LIN {X 0,Y 516.678,Z 319.494,A -85,B 0,C 180,E1 19152.315,E2 19152.315} C_VEL
LIN {X 0,Y 512.908,Z 316.647,A -85,B 0,C 180,E1 19150.24,E2 19150.24} C_VEL
LIN {X 0,Y 508.959,Z 312.336,A -85,B 0,C 180,E1 19148.207,E2 19148.207} C_VEL
LIN {X 0,Y 504.801,Z 309.238,A -85,B 0,C 180,E1 19146.294,E2 19146.294} C_VEL
LIN {X 0,Y 500.678,Z 304.761,A -85,B 0,C 180,E1 19144.449,E2 19144.449} C_VEL
LIN {X 0,Y 496.281,Z 301.328,A -85,B 0,C 180,E1 19142.687,E2 19142.687} C_VEL
LIN {X 0,Y 492.471,Z 297.218,A -85,B 0,C 180,E1 19141.176,E2 19141.176} C_VEL
LIN {X 0,Y 487.825,Z 293.173,A -85,B 0,C 180,E1 19139.452,E2 19139.452} C_VEL
LIN {X 0,Y 484.702,Z 289.843,A -85,B 0,C 180,E1 19138.318,E2 19138.318} C_VEL
LIN {X 0,Y 480.021,Z 285.689,A -85,B 0,C 180,E1 19136.7,E2 19136.7} C_VEL
LIN {X 0,Y 477.029,Z 282.466,A -85,B 0,C 180,E1 19135.676,E2 19135.676} C_VEL
LIN {X 0,Y 472.507,Z 278.285,A -85,B 0,C 180,E1 19134.195,E2 19134.195} C_VEL
LIN {X 0,Y 469.925,Z 275.379,A -85,B 0,C 180,E1 19133.338,E2 19133.338} C_VEL
LIN {X 0,Y 465.029,Z 270.655,A -85,B 0,C 180,E1 19131.803,E2 19131.803} C_VEL
LIN {X 0,Y 462.666,Z 268.183,A -85,B 0,C 180,E1 19131.079,E2 19131.079} C_VEL
LIN {X 0,Y 458.047,Z 263.498,A -85,B 0,C 180,E1 19129.676,E2 19129.676} C_VEL
LIN {X 0,Y 455.814,Z 261.137,A -85,B 0,C 180,E1 19128.992,E2 19128.992} C_VEL
LIN {X 0,Y 451.033,Z 256.164,A -85,B 0,C 180,E1 19127.581,E2 19127.581} C_VEL
LIN {X 0,Y 445.033,Z 249.934,A -85,B 0,C 180,E1 19125.861,E2 19125.861} C_VEL
LIN {X 0,Y 443.054,Z 247.797,A -85,B 0,C 180,E1 19125.308,E2 19125.308} C_VEL
LIN {X 0,Y 438.624,Z 243.367,A -85,B 0,C 180,E1 19124.141,E2 19124.141} C_VEL
LIN {X 0,Y 436.476,Z 241.078,A -85,B 0,C 180,E1 19123.594,E2 19123.594} C_VEL
LIN {X 0,Y 432.178,Z 236.724,A -85,B 0,C 180,E1 19122.544,E2 19122.544} C_VEL
LIN {X 0,Y 430.194,Z 234.427,A -85,B 0,C 180,E1 19122.065,E2 19122.065} C_VEL
LIN {X 0,Y 429.077,Z 233.472,A -85,B 0,C 180,E1 19121.812,E2 19121.812} C_VEL
LIN {X 0,Y 423.316,Z 229.525,A -85,B 0,C 180,E1 19120.566,E2 19120.566} C_VEL
LIN {X 0,Y 413.271,Z 224.33,A -85,B 0,C 180,E1 19118.597,E2 19118.597} C_VEL
LIN {X 0,Y 410.338,Z 222.17,A -85,B 0,C 180,E1 19118.018,E2 19118.018} C_VEL
LIN {X 0,Y 407.486,Z 218.551,A -85,B 0,C 180,E1 19117.396,E2 19117.396} C_VEL
LIN {X 0,Y 406.442,Z 216.882,A -85,B 0,C 180,E1 19117.154,E2 19117.154} C_VEL
LIN {X 0,Y 403.788,Z 214.24,A -85,B 0,C 180,E1 19116.574,E2 19116.574} C_VEL
LIN {X 0,Y 402.666,Z 211.461,A -85,B 0,C 180,E1 19116.164,E2 19116.164} C_VEL
LIN {X 0,Y 402.566,Z 210.942,A -85,B 0,C 180,E1 19115.455,E2 19115.455} C_VEL
LIN {X 0,Y 402.577,Z 211.024,A -85,B 0,C 180,E1 19111.592,E2 19111.592} C_VEL
LIN {X 0,Y 402.567,Z 210.925,A -85,B 0,C 180,E1 19107.676,E2 19107.676} C_VEL
LIN {X 0,Y 402.577,Z 211.022,A -85,B 0,C 180,E1 19103.726,E2 19103.726} C_VEL
LIN {X 0,Y 402.577,Z 211.018,A -85,B 0,C 180,E1 19099.742,E2 19099.742} C_VEL
LIN {X 0,Y 402.573,Z 211.002,A -85,B 0,C 180,E1 19095.856,E2 19095.856} C_VEL
LIN {X 0,Y 402.573,Z 210.991,A -85,B 0,C 180,E1 19091.897,E2 19091.897} C_VEL
LIN {X 0,Y 402.574,Z 210.995,A -85,B 0,C 180,E1 19087.995,E2 19087.995} C_VEL
LIN {X 0,Y 402.574,Z 211.015,A -85,B 0,C 180,E1 19083.988,E2 19083.988} C_VEL
LIN {X 0,Y 402.574,Z 211.02,A -85,B 0,C 180,E1 19080,E2 19080} C_VEL
LIN {X 0,Y 402.574,Z 210.997,A -85,B 0,C 180,E1 19076.012,E2 19076.012} C_VEL
LIN {X 0,Y 402.572,Z 210.987,A -85,B 0,C 180,E1 19072.148,E2 19072.148} C_VEL
LIN {X 0,Y 402.575,Z 211,A -85,B 0,C 180,E1 19068.248,E2 19068.248} C_VEL
LIN {X 0,Y 402.578,Z 211.02,A -85,B 0,C 180,E1 19064.292,E2 19064.292} C_VEL
LIN {X 0,Y 402.579,Z 211.022,A -85,B 0,C 180,E1 19060.409,E2 19060.409} C_VEL
LIN {X 0,Y 402.584,Z 211.009,A -85,B 0,C 180,E1 19056.585,E2 19056.585} C_VEL
LIN {X 0,Y 402.582,Z 210.933,A -85,B 0,C 180,E1 19052.753,E2 19052.753} C_VEL
LIN {X 0,Y 402.591,Z 210.985,A -85,B 0,C 180,E1 19048.896,E2 19048.896} C_VEL
LIN {X 0,Y 402.601,Z 211.025,A -85,B 0,C 180,E1 19045.032,E2 19045.032} C_VEL
LIN {X 0,Y 402.714,Z 211.75,A -85,B 0,C 180,E1 19044.654,E2 19044.654} C_VEL
LIN {X 0,Y 404.399,Z 215.495,A -85,B 0,C 180,E1 19043.6,E2 19043.6} C_VEL
LIN {X 0,Y 414.866,Z 230.627,A -85,B 0,C 180,E1 19041.263,E2 19041.263} C_VEL
LIN {X 0,Y 422.772,Z 242.404,A -85,B 0,C 180,E1 19039.651,E2 19039.651} C_VEL
LIN {X 0,Y 432.944,Z 258.691,A -85,B 0,C 180,E1 19037.706,E2 19037.706} C_VEL
LIN {X 0,Y 444.241,Z 278.519,A -85,B 0,C 180,E1 19035.686,E2 19035.686} C_VEL
LIN {X 0,Y 455.277,Z 300.15,A -85,B 0,C 180,E1 19033.824,E2 19033.824} C_VEL
LIN {X 0,Y 456.625,Z 303.478,A -85,B 0,C 180,E1 19033.592,E2 19033.592} C_VEL
LIN {X 0,Y 447.384,Z 520.785,A -85,B 0,C 180,E1 19030.062,E2 19030.062} C_VEL
LIN {X 0,Y 445.937,Z 538.911,A -85,B 0,C 180,E1 19029.651,E2 19029.651} C_VEL
LIN {X 0,Y 443.556,Z 560.38,A -85,B 0,C 180,E1 19028.986,E2 19028.986} C_VEL
LIN {X 0,Y 440.354,Z 582.229,A -85,B 0,C 180,E1 19028.054,E2 19028.054} C_VEL
LIN {X 0,Y 437.341,Z 599.726,A -85,B 0,C 180,E1 19027.121,E2 19027.121} C_VEL
LIN {X 0,Y 434.267,Z 615.592,A -85,B 0,C 180,E1 19026.111,E2 19026.111} C_VEL
LIN {X 0,Y 431.179,Z 630.152,A -85,B 0,C 180,E1 19025.028,E2 19025.028} C_VEL
LIN {X 0,Y 427.866,Z 644.6,A -85,B 0,C 180,E1 19023.787,E2 19023.787} C_VEL
LIN {X 0,Y 424.501,Z 658.489,A -85,B 0,C 180,E1 19022.412,E2 19022.412} C_VEL
LIN {X 0,Y 421.02,Z 672.173,A -85,B 0,C 180,E1 19020.858,E2 19020.858} C_VEL
LIN {X 0,Y 417.315,Z 686.298,A -85,B 0,C 180,E1 19019.008,E2 19019.008} C_VEL
LIN {X 0,Y 412.921,Z 702.744,A -85,B 0,C 180,E1 19016.455,E2 19016.455} C_VEL
LIN {X 0,Y 409.682,Z 714.914,A -85,B 0,C 180,E1 19014.203,E2 19014.203} C_VEL
LIN {X 0,Y 407.133,Z 724.889,A -85,B 0,C 180,E1 19012.068,E2 19012.068} C_VEL
LIN {X 0,Y 404.954,Z 733.96,A -85,B 0,C 180,E1 19009.822,E2 19009.822} C_VEL
LIN {X 0,Y 403.169,Z 742.134,A -85,B 0,C 180,E1 19007.46,E2 19007.46} C_VEL
LIN {X 0,Y 401.726,Z 749.741,A -85,B 0,C 180,E1 19004.852,E2 19004.852} C_VEL
LIN {X 0,Y 400.599,Z 757.452,A -85,B 0,C 180,E1 19001.517,E2 19001.517} C_VEL
LIN {X 0,Y 400.13,Z 762.218,A -85,B 0,C 180,E1 18998.767,E2 18998.767} C_VEL
LIN {X 0,Y 399.973,Z 765.375,A -85,B 0,C 180,E1 18996.314,E2 18996.314} C_VEL
LIN {X 0,Y 399.939,Z 767.492,A -85,B 0,C 180,E1 18993.87,E2 18993.87} C_VEL
LIN {X 0,Y 399.948,Z 768.59,A -85,B 0,C 180,E1 18991.432,E2 18991.432} C_VEL
LIN {X 0,Y 399.955,Z 768.708,A -85,B 0,C 180,E1 18989.141,E2 18989.141} C_VEL
LIN {X 0,Y 399.936,Z 767.846,A -85,B 0,C 180,E1 18986.704,E2 18986.704} C_VEL
LIN {X 0,Y 399.951,Z 765.967,A -85,B 0,C 180,E1 18984.262,E2 18984.262} C_VEL
LIN {X 0,Y 400.076,Z 762.997,A -85,B 0,C 180,E1 18981.773,E2 18981.773} C_VEL
LIN {X 0,Y 400.407,Z 759.074,A -85,B 0,C 180,E1 18979.352,E2 18979.352} C_VEL
LIN {X 0,Y 401.047,Z 753.989,A -85,B 0,C 180,E1 18976.888,E2 18976.888} C_VEL
LIN {X 0,Y 402.002,Z 748.142,A -85,B 0,C 180,E1 18974.568,E2 18974.568} C_VEL
LIN {X 0,Y 403.361,Z 741.196,A -85,B 0,C 180,E1 18972.25,E2 18972.25} C_VEL
LIN {X 0,Y 405.16,Z 733.067,A -85,B 0,C 180,E1 18969.941,E2 18969.941} C_VEL
LIN {X 0,Y 407.609,Z 723.032,A -85,B 0,C 180,E1 18967.504,E2 18967.504} C_VEL
LIN {X 0,Y 411.234,Z 709.077,A -85,B 0,C 180,E1 18964.667,E2 18964.667} C_VEL
LIN {X 0,Y 414.498,Z 696.788,A -85,B 0,C 180,E1 18962.569,E2 18962.569} C_VEL
LIN {X 0,Y 417.854,Z 684.221,A -85,B 0,C 180,E1 18960.706,E2 18960.706} C_VEL
LIN {X 0,Y 421.097,Z 671.876,A -85,B 0,C 180,E1 18959.106,E2 18959.106} C_VEL
LIN {X 0,Y 424.501,Z 658.492,A -85,B 0,C 180,E1 18957.588,E2 18957.588} C_VEL
LIN {X 0,Y 427.867,Z 644.6,A -85,B 0,C 180,E1 18956.213,E2 18956.213} C_VEL
LIN {X 0,Y 431.179,Z 630.151,A -85,B 0,C 180,E1 18954.972,E2 18954.972} C_VEL
LIN {X 0,Y 434.454,Z 614.671,A -85,B 0,C 180,E1 18953.825,E2 18953.825} C_VEL
LIN {X 0,Y 437.539,Z 598.663,A -85,B 0,C 180,E1 18952.817,E2 18952.817} C_VEL
LIN {X 0,Y 440.807,Z 579.508,A -85,B 0,C 180,E1 18951.812,E2 18951.812} C_VEL
LIN {X 0,Y 443.971,Z 556.629,A -85,B 0,C 180,E1 18950.887,E2 18950.887} C_VEL
LIN {X 0,Y 446.015,Z 538.025,A -85,B 0,C 180,E1 18950.326,E2 18950.326} C_VEL
LIN {X 0,Y 447.414,Z 520.27,A -85,B 0,C 180,E1 18949.928,E2 18949.928} C_VEL
LIN {X 0,Y 456.615,Z 302.923,A -85,B 0,C 180,E1 18946.395,E2 18946.395} C_VEL
LIN {X 0,Y 445.675,Z 281.186,A -85,B 0,C 180,E1 18944.561,E2 18944.561} C_VEL
LIN {X 0,Y 434.191,Z 260.787,A -85,B 0,C 180,E1 18942.524,E2 18942.524} C_VEL
LIN {X 0,Y 424.621,Z 245.292,A -85,B 0,C 180,E1 18940.714,E2 18940.714} C_VEL
LIN {X 0,Y 416.039,Z 232.351,A -85,B 0,C 180,E1 18938.983,E2 18938.983} C_VEL
LIN {X 0,Y 408.694,Z 221.675,A -85,B 0,C 180,E1 18937.399,E2 18937.399} C_VEL
LIN {X 0,Y 404.615,Z 215.942,A -85,B 0,C 180,E1 18936.465,E2 18936.465} C_VEL
LIN {X 0,Y 403.803,Z 214.337,A -85,B 0,C 180,E1 18936.11,E2 18936.11} C_VEL
LIN {X 0,Y 402.6,Z 211.068,A -85,B 0,C 180,E1 18935.09,E2 18935.09} C_VEL
LIN {X 0,Y 402.583,Z 210.994,A -85,B 0,C 180,E1 18931.272,E2 18931.272} C_VEL
LIN {X 0,Y 402.571,Z 210.93,A -85,B 0,C 180,E1 18927.515,E2 18927.515} C_VEL
LIN {X 0,Y 402.578,Z 211.013,A -85,B 0,C 180,E1 18923.6,E2 18923.6} C_VEL
LIN {X 0,Y 402.577,Z 211.019,A -85,B 0,C 180,E1 18919.742,E2 18919.742} C_VEL
LIN {X 0,Y 402.576,Z 211.012,A -85,B 0,C 180,E1 18915.856,E2 18915.856} C_VEL
LIN {X 0,Y 402.575,Z 210.997,A -85,B 0,C 180,E1 18911.897,E2 18911.897} C_VEL
LIN {X 0,Y 402.574,Z 210.989,A -85,B 0,C 180,E1 18907.995,E2 18907.995} C_VEL
LIN {X 0,Y 402.577,Z 211.003,A -85,B 0,C 180,E1 18904.131,E2 18904.131} C_VEL
LIN {X 0,Y 402.579,Z 211.021,A -85,B 0,C 180,E1 18900.285,E2 18900.285} C_VEL
LIN {X 0,Y 402.583,Z 211.003,A -85,B 0,C 180,E1 18896.44,E2 18896.44} C_VEL
LIN {X 0,Y 402.587,Z 210.991,A -85,B 0,C 180,E1 18892.58,E2 18892.58} C_VEL
LIN {X 0,Y 402.599,Z 210.996,A -85,B 0,C 180,E1 18888.779,E2 18888.779} C_VEL
LIN {X 0,Y 402.606,Z 211.014,A -85,B 0,C 180,E1 18884.884,E2 18884.884} C_VEL
LIN {X 0,Y 402.614,Z 211.016,A -85,B 0,C 180,E1 18881.014,E2 18881.014} C_VEL
LIN {X 0,Y 402.614,Z 211.007,A -85,B 0,C 180,E1 18877.051,E2 18877.051} C_VEL
LIN {X 0,Y 402.603,Z 210.927,A -85,B 0,C 180,E1 18873.127,E2 18873.127} C_VEL
LIN {X 0,Y 402.619,Z 210.988,A -85,B 0,C 180,E1 18869.222,E2 18869.222} C_VEL
LIN {X 0,Y 402.607,Z 210.937,A -85,B 0,C 180,E1 18865.279,E2 18865.279} C_VEL
LIN {X 0,Y 402.629,Z 211.28,A -85,B 0,C 180,E1 18863.91,E2 18863.91} C_VEL
LIN {X 0,Y 403.059,Z 212.799,A -85,B 0,C 180,E1 18863.615,E2 18863.615} C_VEL
LIN {X 0,Y 405.049,Z 215.794,A -85,B 0,C 180,E1 18863.14,E2 18863.14} C_VEL
LIN {X 0,Y 407.043,Z 217.67,A -85,B 0,C 180,E1 18862.711,E2 18862.711} C_VEL
LIN {X 0,Y 409.632,Z 221.504,A -85,B 0,C 180,E1 18862.128,E2 18862.128} C_VEL
LIN {X 0,Y 411.583,Z 223.575,A -85,B 0,C 180,E1 18861.721,E2 18861.721} C_VEL
LIN {X 0,Y 414.872,Z 227.805,A -85,B 0,C 180,E1 18861.02,E2 18861.02} C_VEL
LIN {X 0,Y 416.966,Z 229.994,A -85,B 0,C 180,E1 18860.589,E2 18860.589} C_VEL
LIN {X 0,Y 420.872,Z 234.538,A -85,B 0,C 180,E1 18859.744,E2 18859.744} C_VEL
LIN {X 0,Y 423.013,Z 236.84,A -85,B 0,C 180,E1 18859.278,E2 18859.278} C_VEL
LIN {X 0,Y 427.436,Z 241.517,A -85,B 0,C 180,E1 18858.277,E2 18858.277} C_VEL
LIN {X 0,Y 433.186,Z 247.672,A -85,B 0,C 180,E1 18856.903,E2 18856.903} C_VEL
LIN {X 0,Y 435.865,Z 250.266,A -85,B 0,C 180,E1 18856.248,E2 18856.248} C_VEL
LIN {X 0,Y 440.63,Z 255.029,A -85,B 0,C 180,E1 18855.019,E2 18855.019} C_VEL
LIN {X 0,Y 443.473,Z 258.126,A -85,B 0,C 180,E1 18854.24,E2 18854.24} C_VEL
LIN {X 0,Y 449.145,Z 263.898,A -85,B 0,C 180,E1 18852.628,E2 18852.628} C_VEL
LIN {X 0,Y 454.171,Z 268.914,A -85,B 0,C 180,E1 18851.154,E2 18851.154} C_VEL
LIN {X 0,Y 460.431,Z 275.421,A -85,B 0,C 180,E1 18849.268,E2 18849.268} C_VEL
LIN {X 0,Y 463.074,Z 278.17,A -85,B 0,C 180,E1 18848.446,E2 18848.446} C_VEL
LIN {X 0,Y 468.112,Z 282.967,A -85,B 0,C 180,E1 18846.88,E2 18846.88} C_VEL
LIN {X 0,Y 473.992,Z 289.045,A -85,B 0,C 180,E1 18844.971,E2 18844.971} C_VEL
LIN {X 0,Y 476.782,Z 291.54,A -85,B 0,C 180,E1 18844.047,E2 18844.047} C_VEL
LIN {X 0,Y 481.738,Z 296.473,A -85,B 0,C 180,E1 18842.353,E2 18842.353} C_VEL
LIN {X 0,Y 484.411,Z 298.833,A -85,B 0,C 180,E1 18841.403,E2 18841.403} C_VEL
LIN {X 0,Y 489.55,Z 303.886,A -85,B 0,C 180,E1 18839.53,E2 18839.53} C_VEL
LIN {X 0,Y 492.121,Z 306.093,A -85,B 0,C 180,E1 18838.553,E2 18838.553} C_VEL
LIN {X 0,Y 496.703,Z 310.742,A -85,B 0,C 180,E1 18836.734,E2 18836.734} C_VEL
LIN {X 0,Y 500.151,Z 313.415,A -85,B 0,C 180,E1 18835.326,E2 18835.326} C_VEL
LIN {X 0,Y 504.25,Z 317.738,A -85,B 0,C 180,E1 18833.485,E2 18833.485} C_VEL
LIN {X 0,Y 508.547,Z 320.982,A -85,B 0,C 180,E1 18831.504,E2 18831.504} C_VEL
LIN {X 0,Y 512.494,Z 325.24,A -85,B 0,C 180,E1 18829.427,E2 18829.427} C_VEL
LIN {X 0,Y 516.343,Z 327.806,A -85,B 0,C 180,E1 18827.313,E2 18827.313} C_VEL
LIN {X 0,Y 517.373,Z 328.757,A -85,B 0,C 180,E1 18826.676,E2 18826.676} C_VEL
LIN {X 0,Y 520.319,Z 332.194,A -85,B 0,C 180,E1 18824.692,E2 18824.692} C_VEL
LIN {X 0,Y 523.276,Z 334.471,A -85,B 0,C 180,E1 18822.463,E2 18822.463} C_VEL
LIN {X 0,Y 526.397,Z 336.084,A -85,B 0,C 180,E1 18819.732,E2 18819.732} C_VEL
LIN {X 0,Y 528.008,Z 338.572,A -85,B 0,C 180,E1 18817.726,E2 18817.726} C_VEL
LIN {X 0,Y 529.556,Z 340.281,A -85,B 0,C 180,E1 18815.308,E2 18815.308} C_VEL
LIN {X 0,Y 530.568,Z 341.191,A -85,B 0,C 180,E1 18812.7,E2 18812.7} C_VEL
LIN {X 0,Y 530.957,Z 341.428,A -85,B 0,C 180,E1 18810.108,E2 18810.108} C_VEL
LIN {X 0,Y 530.628,Z 341.205,A -85,B 0,C 180,E1 18807.516,E2 18807.516} C_VEL
LIN {X 0,Y 529.697,Z 340.427,A -85,B 0,C 180,E1 18805.019,E2 18805.019} C_VEL
LIN {X 0,Y 528.245,Z 338.827,A -85,B 0,C 180,E1 18802.606,E2 18802.606} C_VEL
LIN {X 0,Y 526.785,Z 336.773,A -85,B 0,C 180,E1 18800.717,E2 18800.717} C_VEL
LIN {X 0,Y 525.736,Z 335.636,A -85,B 0,C 180,E1 18799.592,E2 18799.592} C_VEL
LIN {X 0,Y 522.885,Z 334.219,A -85,B 0,C 180,E1 18797.227,E2 18797.227} C_VEL
LIN {X 0,Y 519.79,Z 331.689,A -85,B 0,C 180,E1 18794.95,E2 18794.95} C_VEL
LIN {X 0,Y 517.018,Z 328.198,A -85,B 0,C 180,E1 18793.081,E2 18793.081} C_VEL
LIN {X 0,Y 512.848,Z 325.533,A -85,B 0,C 180,E1 18790.765,E2 18790.765} C_VEL
LIN {X 0,Y 509.073,Z 321.621,A -85,B 0,C 180,E1 18788.756,E2 18788.756} C_VEL
LIN {X 0,Y 507.542,Z 320.084,A -85,B 0,C 180,E1 18788.021,E2 18788.021} C_VEL
LIN {X 0,Y 503.184,Z 316.758,A -85,B 0,C 180,E1 18786.021,E2 18786.021} C_VEL
LIN {X 0,Y 499.095,Z 312.438,A -85,B 0,C 180,E1 18784.235,E2 18784.235} C_VEL
LIN {X 0,Y 494.737,Z 308.992,A -85,B 0,C 180,E1 18782.491,E2 18782.491} C_VEL
LIN {X 0,Y 490.774,Z 304.808,A -85,B 0,C 180,E1 18780.931,E2 18780.931} C_VEL
LIN {X 0,Y 485.858,Z 300.436,A -85,B 0,C 180,E1 18779.113,E2 18779.113} C_VEL
LIN {X 0,Y 482.799,Z 297.305,A -85,B 0,C 180,E1 18778.022,E2 18778.022} C_VEL
LIN {X 0,Y 477.809,Z 292.72,A -85,B 0,C 180,E1 18776.299,E2 18776.299} C_VEL
LIN {X 0,Y 475.019,Z 289.871,A -85,B 0,C 180,E1 18775.371,E2 18775.371} C_VEL
LIN {X 0,Y 470.307,Z 285.411,A -85,B 0,C 180,E1 18773.834,E2 18773.834} C_VEL
LIN {X 0,Y 467.682,Z 282.64,A -85,B 0,C 180,E1 18772.99,E2 18772.99} C_VEL
LIN {X 0,Y 462.77,Z 277.812,A -85,B 0,C 180,E1 18771.459,E2 18771.459} C_VEL
LIN {X 0,Y 460.22,Z 275.239,A -85,B 0,C 180,E1 18770.666,E2 18770.666} C_VEL
LIN {X 0,Y 455.157,Z 269.84,A -85,B 0,C 180,E1 18769.13,E2 18769.13} C_VEL
LIN {X 0,Y 449.254,Z 264.034,A -85,B 0,C 180,E1 18767.404,E2 18767.404} C_VEL
LIN {X 0,Y 446.709,Z 261.397,A -85,B 0,C 180,E1 18766.674,E2 18766.674} C_VEL
LIN {X 0,Y 442.141,Z 256.472,A -85,B 0,C 180,E1 18765.382,E2 18765.382} C_VEL
LIN {X 0,Y 436.243,Z 250.726,A -85,B 0,C 180,E1 18763.85,E2 18763.85} C_VEL
LIN {X 0,Y 433.693,Z 248.089,A -85,B 0,C 180,E1 18763.215,E2 18763.215} C_VEL
LIN {X 0,Y 429.082,Z 243.341,A -85,B 0,C 180,E1 18762.109,E2 18762.109} C_VEL
LIN {X 0,Y 423.013,Z 236.84,A -85,B 0,C 180,E1 18760.722,E2 18760.722} C_VEL
LIN {X 0,Y 420.872,Z 234.537,A -85,B 0,C 180,E1 18760.256,E2 18760.256} C_VEL
LIN {X 0,Y 416.966,Z 229.993,A -85,B 0,C 180,E1 18759.411,E2 18759.411} C_VEL
LIN {X 0,Y 412.115,Z 224.465,A -85,B 0,C 180,E1 18758.398,E2 18758.398} C_VEL
LIN {X 0,Y 410.618,Z 222.406,A -85,B 0,C 180,E1 18758.075,E2 18758.075} C_VEL
LIN {X 0,Y 410.338,Z 222.17,A -85,B 0,C 180,E1 18758.018,E2 18758.018} C_VEL
LIN {X 0,Y 406.6,Z 220.205,A -85,B 0,C 180,E1 18757.279,E2 18757.279} C_VEL
LIN {X 0,Y 398.861,Z 218.042,A -85,B 0,C 180,E1 18755.719,E2 18755.719} C_VEL
LIN {X 0,Y 396.986,Z 216.669,A -85,B 0,C 180,E1 18755.296,E2 18755.296} C_VEL
LIN {X 0,Y 395.077,Z 213.661,A -85,B 0,C 180,E1 18754.8,E2 18754.8} C_VEL
LIN {X 0,Y 394.701,Z 212.186,A -85,B 0,C 180,E1 18754.48,E2 18754.48} C_VEL
LIN {X 0,Y 394.678,Z 211.963,A -85,B 0,C 180,E1 18750.543,E2 18750.543} C_VEL
LIN {X 0,Y 394.668,Z 211.917,A -85,B 0,C 180,E1 18746.594,E2 18746.594} C_VEL
LIN {X 0,Y 394.682,Z 211.988,A -85,B 0,C 180,E1 18742.649,E2 18742.649} C_VEL
LIN {X 0,Y 394.674,Z 211.997,A -85,B 0,C 180,E1 18738.616,E2 18738.616} C_VEL
LIN {X 0,Y 394.67,Z 212.005,A -85,B 0,C 180,E1 18734.612,E2 18734.612} C_VEL
LIN {X 0,Y 394.665,Z 211.993,A -85,B 0,C 180,E1 18730.621,E2 18730.621} C_VEL
LIN {X 0,Y 394.666,Z 211.978,A -85,B 0,C 180,E1 18726.693,E2 18726.693} C_VEL
LIN {X 0,Y 394.665,Z 211.976,A -85,B 0,C 180,E1 18722.759,E2 18722.759} C_VEL
LIN {X 0,Y 394.675,Z 211.996,A -85,B 0,C 180,E1 18718.839,E2 18718.839} C_VEL
LIN {X 0,Y 394.673,Z 212.001,A -85,B 0,C 180,E1 18714.913,E2 18714.913} C_VEL
LIN {X 0,Y 394.673,Z 211.979,A -85,B 0,C 180,E1 18710.963,E2 18710.963} C_VEL
LIN {X 0,Y 394.671,Z 211.976,A -85,B 0,C 180,E1 18706.969,E2 18706.969} C_VEL
LIN {X 0,Y 394.675,Z 211.98,A -85,B 0,C 180,E1 18703.061,E2 18703.061} C_VEL
LIN {X 0,Y 394.677,Z 211.989,A -85,B 0,C 180,E1 18699.071,E2 18699.071} C_VEL
LIN {X 0,Y 394.676,Z 211.993,A -85,B 0,C 180,E1 18695.13,E2 18695.13} C_VEL
LIN {X 0,Y 394.674,Z 211.91,A -85,B 0,C 180,E1 18691.218,E2 18691.218} C_VEL
LIN {X 0,Y 394.677,Z 211.984,A -85,B 0,C 180,E1 18687.244,E2 18687.244} C_VEL
LIN {X 0,Y 394.688,Z 212.311,A -85,B 0,C 180,E1 18686.128,E2 18686.128} C_VEL
LIN {X 0,Y 395.717,Z 215.02,A -85,B 0,C 180,E1 18685.352,E2 18685.352} C_VEL
LIN {X 0,Y 400.359,Z 221.234,A -85,B 0,C 180,E1 18684.194,E2 18684.194} C_VEL
LIN {X 0,Y 411.418,Z 237.249,A -85,B 0,C 180,E1 18681.68,E2 18681.68} C_VEL
LIN {X 0,Y 419.024,Z 248.756,A -85,B 0,C 180,E1 18680.089,E2 18680.089} C_VEL
LIN {X 0,Y 428.723,Z 264.464,A -85,B 0,C 180,E1 18678.184,E2 18678.184} C_VEL
LIN {X 0,Y 439.743,Z 284.053,A -85,B 0,C 180,E1 18676.159,E2 18676.159} C_VEL
LIN {X 0,Y 450.503,Z 305.432,A -85,B 0,C 180,E1 18674.292,E2 18674.292} C_VEL
LIN {X 0,Y 450.665,Z 307.342,A -85,B 0,C 180,E1 18674.23,E2 18674.23} C_VEL
LIN {X 0,Y 441.27,Z 520.712,A -85,B 0,C 180,E1 18670.73,E2 18670.73} C_VEL
LIN {X 0,Y 439.762,Z 539.03,A -85,B 0,C 180,E1 18670.31,E2 18670.31} C_VEL
LIN {X 0,Y 437.286,Z 560.653,A -85,B 0,C 180,E1 18669.633,E2 18669.633} C_VEL
LIN {X 0,Y 434.042,Z 582.053,A -85,B 0,C 180,E1 18668.709,E2 18668.709} C_VEL
LIN {X 0,Y 430.937,Z 599.55,A -85,B 0,C 180,E1 18667.768,E2 18667.768} C_VEL
LIN {X 0,Y 427.763,Z 615.416,A -85,B 0,C 180,E1 18666.749,E2 18666.749} C_VEL
LIN {X 0,Y 424.372,Z 630.861,A -85,B 0,C 180,E1 18665.584,E2 18665.584} C_VEL
LIN {X 0,Y 420.802,Z 645.845,A -85,B 0,C 180,E1 18664.268,E2 18664.268} C_VEL
LIN {X 0,Y 416.794,Z 661.744,A -85,B 0,C 180,E1 18662.642,E2 18662.642} C_VEL
LIN {X 0,Y 411.865,Z 680.047,A -85,B 0,C 180,E1 18660.405,E2 18660.405} C_VEL
LIN {X 0,Y 408.258,Z 693.05,A -85,B 0,C 180,E1 18658.524,E2 18658.524} C_VEL
LIN {X 0,Y 404.944,Z 704.94,A -85,B 0,C 180,E1 18656.543,E2 18656.543} C_VEL
LIN {X 0,Y 402.043,Z 715.437,A -85,B 0,C 180,E1 18654.537,E2 18654.537} C_VEL
LIN {X 0,Y 399.402,Z 725.329,A -85,B 0,C 180,E1 18652.363,E2 18652.363} C_VEL
LIN {X 0,Y 397.172,Z 734.199,A -85,B 0,C 180,E1 18650.109,E2 18650.109} C_VEL
LIN {X 0,Y 395.289,Z 742.424,A -85,B 0,C 180,E1 18647.668,E2 18647.668} C_VEL
LIN {X 0,Y 393.595,Z 751.154,A -85,B 0,C 180,E1 18644.557,E2 18644.557} C_VEL
LIN {X 0,Y 392.583,Z 757.815,A -85,B 0,C 180,E1 18641.457,E2 18641.457} C_VEL
LIN {X 0,Y 392.145,Z 762.042,A -85,B 0,C 180,E1 18638.947,E2 18638.947} C_VEL
LIN {X 0,Y 391.976,Z 765.199,A -85,B 0,C 180,E1 18636.444,E2 18636.444} C_VEL
LIN {X 0,Y 391.939,Z 767.317,A -85,B 0,C 180,E1 18633.949,E2 18633.949} C_VEL
LIN {X 0,Y 391.95,Z 768.415,A -85,B 0,C 180,E1 18631.462,E2 18631.462} C_VEL
LIN {X 0,Y 391.957,Z 768.533,A -85,B 0,C 180,E1 18629.123,E2 18629.123} C_VEL
LIN {X 0,Y 391.937,Z 767.671,A -85,B 0,C 180,E1 18626.637,E2 18626.637} C_VEL
LIN {X 0,Y 391.956,Z 765.791,A -85,B 0,C 180,E1 18624.144,E2 18624.144} C_VEL
LIN {X 0,Y 392.089,Z 762.876,A -85,B 0,C 180,E1 18621.643,E2 18621.643} C_VEL
LIN {X 0,Y 392.451,Z 758.897,A -85,B 0,C 180,E1 18619.134,E2 18619.134} C_VEL
LIN {X 0,Y 393.134,Z 753.811,A -85,B 0,C 180,E1 18616.62,E2 18616.62} C_VEL
LIN {X 0,Y 394.151,Z 747.964,A -85,B 0,C 180,E1 18614.252,E2 18614.252} C_VEL
LIN {X 0,Y 395.605,Z 740.95,A -85,B 0,C 180,E1 18611.868,E2 18611.868} C_VEL
LIN {X 0,Y 397.49,Z 732.889,A -85,B 0,C 180,E1 18609.537,E2 18609.537} C_VEL
LIN {X 0,Y 399.895,Z 723.473,A -85,B 0,C 180,E1 18607.201,E2 18607.201} C_VEL
LIN {X 0,Y 403.495,Z 710.304,A -85,B 0,C 180,E1 18604.426,E2 18604.426} C_VEL
LIN {X 0,Y 407.269,Z 696.61,A -85,B 0,C 180,E1 18602.04,E2 18602.04} C_VEL
LIN {X 0,Y 410.758,Z 684.043,A -85,B 0,C 180,E1 18600.15,E2 18600.15} C_VEL
LIN {X 0,Y 414.197,Z 671.434,A -85,B 0,C 180,E1 18598.495,E2 18598.495} C_VEL
LIN {X 0,Y 417.791,Z 657.798,A -85,B 0,C 180,E1 18596.935,E2 18596.935} C_VEL
LIN {X 0,Y 421.275,Z 643.884,A -85,B 0,C 180,E1 18595.548,E2 18595.548} C_VEL
LIN {X 0,Y 424.738,Z 629.249,A -85,B 0,C 180,E1 18594.286,E2 18594.286} C_VEL
LIN {X 0,Y 428.15,Z 613.574,A -85,B 0,C 180,E1 18593.122,E2 18593.122} C_VEL
LIN {X 0,Y 431.902,Z 594.567,A -85,B 0,C 180,E1 18591.937,E2 18591.937} C_VEL
LIN {X 0,Y 435.519,Z 572.62,A -85,B 0,C 180,E1 18590.856,E2 18590.856} C_VEL
LIN {X 0,Y 438.03,Z 554.255,A -85,B 0,C 180,E1 18590.15,E2 18590.15} C_VEL
LIN {X 0,Y 439.981,Z 536.67,A -85,B 0,C 180,E1 18589.629,E2 18589.629} C_VEL
LIN {X 0,Y 441.375,Z 518.965,A -85,B 0,C 180,E1 18589.236,E2 18589.236} C_VEL
LIN {X 0,Y 450.655,Z 305.754,A -85,B 0,C 180,E1 18585.734,E2 18585.734} C_VEL
LIN {X 0,Y 439.965,Z 284.481,A -85,B 0,C 180,E1 18583.881,E2 18583.881} C_VEL
LIN {X 0,Y 428.939,Z 264.843,A -85,B 0,C 180,E1 18581.857,E2 18581.857} C_VEL
LIN {X 0,Y 419.935,Z 250.22,A -85,B 0,C 180,E1 18580.097,E2 18580.097} C_VEL
LIN {X 0,Y 412.03,Z 238.164,A -85,B 0,C 180,E1 18578.452,E2 18578.452} C_VEL
LIN {X 0,Y 403.996,Z 226.444,A -85,B 0,C 180,E1 18576.662,E2 18576.662} C_VEL
LIN {X 0,Y 399.695,Z 220.552,A -85,B 0,C 180,E1 18575.654,E2 18575.654} C_VEL
LIN {X 0,Y 395.543,Z 214.711,A -85,B 0,C 180,E1 18574.577,E2 18574.577} C_VEL
LIN {X 0,Y 394.651,Z 212.086,A -85,B 0,C 180,E1 18573.757,E2 18573.757} C_VEL
LIN {X 0,Y 394.631,Z 211.93,A -85,B 0,C 180,E1 18569.776,E2 18569.776} C_VEL
LIN {X 0,Y 394.635,Z 211.957,A -85,B 0,C 180,E1 18565.836,E2 18565.836} C_VEL
LIN {X 0,Y 394.64,Z 211.982,A -85,B 0,C 180,E1 18561.998,E2 18561.998} C_VEL
LIN {X 0,Y 394.646,Z 211.98,A -85,B 0,C 180,E1 18558.158,E2 18558.158} C_VEL
LIN {X 0,Y 394.644,Z 211.99,A -85,B 0,C 180,E1 18554.227,E2 18554.227} C_VEL
LIN {X 0,Y 394.65,Z 212.006,A -85,B 0,C 180,E1 18550.363,E2 18550.363} C_VEL
LIN {X 0,Y 394.657,Z 211.99,A -85,B 0,C 180,E1 18546.547,E2 18546.547} C_VEL
LIN {X 0,Y 394.657,Z 211.978,A -85,B 0,C 180,E1 18542.614,E2 18542.614} C_VEL
LIN {X 0,Y 394.661,Z 211.981,A -85,B 0,C 180,E1 18538.693,E2 18538.693} C_VEL
LIN {X 0,Y 394.664,Z 212.003,A -85,B 0,C 180,E1 18534.767,E2 18534.767} C_VEL
LIN {X 0,Y 394.677,Z 211.998,A -85,B 0,C 180,E1 18530.963,E2 18530.963} C_VEL
LIN {X 0,Y 394.671,Z 211.981,A -85,B 0,C 180,E1 18526.969,E2 18526.969} C_VEL
LIN {X 0,Y 394.674,Z 211.978,A -85,B 0,C 180,E1 18523.061,E2 18523.061} C_VEL
LIN {X 0,Y 394.676,Z 211.982,A -85,B 0,C 180,E1 18519.071,E2 18519.071} C_VEL
LIN {X 0,Y 394.672,Z 211.969,A -85,B 0,C 180,E1 18515.13,E2 18515.13} C_VEL
LIN {X 0,Y 394.675,Z 211.914,A -85,B 0,C 180,E1 18511.218,E2 18511.218} C_VEL
LIN {X 0,Y 394.674,Z 211.965,A -85,B 0,C 180,E1 18507.245,E2 18507.245} C_VEL
LIN {X 0,Y 394.714,Z 212.269,A -85,B 0,C 180,E1 18505.516,E2 18505.516} C_VEL
LIN {X 0,Y 395.129,Z 213.801,A -85,B 0,C 180,E1 18505.183,E2 18505.183} C_VEL
LIN {X 0,Y 397.036,Z 216.718,A -85,B 0,C 180,E1 18504.692,E2 18504.692} C_VEL
LIN {X 0,Y 399.239,Z 218.586,A -85,B 0,C 180,E1 18504.189,E2 18504.189} C_VEL
LIN {X 0,Y 401.723,Z 222.397,A -85,B 0,C 180,E1 18503.585,E2 18503.585} C_VEL
LIN {X 0,Y 403.741,Z 224.553,A -85,B 0,C 180,E1 18503.134,E2 18503.134} C_VEL
LIN {X 0,Y 406.943,Z 228.795,A -85,B 0,C 180,E1 18502.413,E2 18502.413} C_VEL
LIN {X 0,Y 412.182,Z 235.086,A -85,B 0,C 180,E1 18501.298,E2 18501.298} C_VEL
LIN {X 0,Y 417.972,Z 241.58,A -85,B 0,C 180,E1 18500.08,E2 18500.08} C_VEL
LIN {X 0,Y 424.381,Z 248.368,A -85,B 0,C 180,E1 18498.677,E2 18498.677} C_VEL
LIN {X 0,Y 430.742,Z 254.975,A -85,B 0,C 180,E1 18497.19,E2 18497.19} C_VEL
LIN {X 0,Y 433.742,Z 257.935,A -85,B 0,C 180,E1 18496.473,E2 18496.473} C_VEL
LIN {X 0,Y 438.9,Z 262.817,A -85,B 0,C 180,E1 18495.163,E2 18495.163} C_VEL
LIN {X 0,Y 444.478,Z 268.704,A -85,B 0,C 180,E1 18493.635,E2 18493.635} C_VEL
LIN {X 0,Y 447.408,Z 271.795,A -85,B 0,C 180,E1 18492.789,E2 18492.789} C_VEL
LIN {X 0,Y 453.976,Z 278.38,A -85,B 0,C 180,E1 18490.874,E2 18490.874} C_VEL
LIN {X 0,Y 459.331,Z 283.595,A -85,B 0,C 180,E1 18489.269,E2 18489.269} C_VEL
LIN {X 0,Y 465.019,Z 289.531,A -85,B 0,C 180,E1 18487.493,E2 18487.493} C_VEL
LIN {X 0,Y 467.754,Z 292.118,A -85,B 0,C 180,E1 18486.642,E2 18486.642} C_VEL
LIN {X 0,Y 472.674,Z 296.992,A -85,B 0,C 180,E1 18485.049,E2 18485.049} C_VEL
LIN {X 0,Y 475.178,Z 299.345,A -85,B 0,C 180,E1 18484.211,E2 18484.211} C_VEL
LIN {X 0,Y 480.261,Z 304.273,A -85,B 0,C 180,E1 18482.485,E2 18482.485} C_VEL
LIN {X 0,Y 482.883,Z 306.638,A -85,B 0,C 180,E1 18481.561,E2 18481.561} C_VEL
LIN {X 0,Y 488.042,Z 311.618,A -85,B 0,C 180,E1 18479.694,E2 18479.694} C_VEL
LIN {X 0,Y 490.695,Z 313.956,A -85,B 0,C 180,E1 18478.689,E2 18478.689} C_VEL
LIN {X 0,Y 495.373,Z 318.573,A -85,B 0,C 180,E1 18476.854,E2 18476.854} C_VEL
LIN {X 0,Y 498.789,Z 321.253,A -85,B 0,C 180,E1 18475.466,E2 18475.466} C_VEL
LIN {X 0,Y 503.102,Z 325.685,A -85,B 0,C 180,E1 18473.542,E2 18473.542} C_VEL
LIN {X 0,Y 507.255,Z 328.839,A -85,B 0,C 180,E1 18471.627,E2 18471.627} C_VEL
LIN {X 0,Y 511.324,Z 333.121,A -85,B 0,C 180,E1 18469.516,E2 18469.516} C_VEL
LIN {X 0,Y 515.21,Z 335.698,A -85,B 0,C 180,E1 18467.388,E2 18467.388} C_VEL
LIN {X 0,Y 516.305,Z 336.8,A -85,B 0,C 180,E1 18466.711,E2 18466.711} C_VEL
LIN {X 0,Y 519.282,Z 340.155,A -85,B 0,C 180,E1 18464.722,E2 18464.722} C_VEL
LIN {X 0,Y 522.274,Z 342.42,A -85,B 0,C 180,E1 18462.474,E2 18462.474} C_VEL
LIN {X 0,Y 525.283,Z 343.929,A -85,B 0,C 180,E1 18459.863,E2 18459.863} C_VEL
LIN {X 0,Y 526.932,Z 346.432,A -85,B 0,C 180,E1 18457.852,E2 18457.852} C_VEL
LIN {X 0,Y 528.421,Z 348.114,A -85,B 0,C 180,E1 18455.537,E2 18455.537} C_VEL
LIN {X 0,Y 529.539,Z 349.101,A -85,B 0,C 180,E1 18452.922,E2 18452.922} C_VEL
LIN {X 0,Y 529.938,Z 349.365,A -85,B 0,C 180,E1 18450.432,E2 18450.432} C_VEL
LIN {X 0,Y 529.729,Z 349.18,A -85,B 0,C 180,E1 18447.837,E2 18447.837} C_VEL
LIN {X 0,Y 528.856,Z 348.505,A -85,B 0,C 180,E1 18445.337,E2 18445.337} C_VEL
LIN {X 0,Y 527.485,Z 347.065,A -85,B 0,C 180,E1 18442.923,E2 18442.923} C_VEL
LIN {X 0,Y 525.874,Z 344.934,A -85,B 0,C 180,E1 18440.811,E2 18440.811} C_VEL
LIN {X 0,Y 524.845,Z 343.621,A -85,B 0,C 180,E1 18439.685,E2 18439.685} C_VEL
LIN {X 0,Y 522.102,Z 342.311,A -85,B 0,C 180,E1 18437.391,E2 18437.391} C_VEL
LIN {X 0,Y 519.107,Z 339.993,A -85,B 0,C 180,E1 18435.159,E2 18435.159} C_VEL
LIN {X 0,Y 516.103,Z 336.5,A -85,B 0,C 180,E1 18433.151,E2 18433.151} C_VEL
LIN {X 0,Y 514.768,Z 335.471,A -85,B 0,C 180,E1 18432.364,E2 18432.364} C_VEL
LIN {X 0,Y 510.721,Z 332.573,A -85,B 0,C 180,E1 18430.146,E2 18430.146} C_VEL
LIN {X 0,Y 506.13,Z 327.83,A -85,B 0,C 180,E1 18427.835,E2 18427.835} C_VEL
LIN {X 0,Y 501.545,Z 324.283,A -85,B 0,C 180,E1 18425.756,E2 18425.756} C_VEL
LIN {X 0,Y 497.52,Z 320.11,A -85,B 0,C 180,E1 18424.02,E2 18424.02} C_VEL
LIN {X 0,Y 493.147,Z 316.604,A -85,B 0,C 180,E1 18422.273,E2 18422.273} C_VEL
LIN {X 0,Y 489.078,Z 312.393,A -85,B 0,C 180,E1 18420.687,E2 18420.687} C_VEL
LIN {X 0,Y 483.916,Z 307.776,A -85,B 0,C 180,E1 18418.807,E2 18418.807} C_VEL
LIN {X 0,Y 481.048,Z 304.866,A -85,B 0,C 180,E1 18417.777,E2 18417.777} C_VEL
LIN {X 0,Y 475.742,Z 299.987,A -85,B 0,C 180,E1 18415.978,E2 18415.978} C_VEL
LIN {X 0,Y 473.305,Z 297.489,A -85,B 0,C 180,E1 18415.159,E2 18415.159} C_VEL
LIN {X 0,Y 468.231,Z 292.683,A -85,B 0,C 180,E1 18413.514,E2 18413.514} C_VEL
LIN {X 0,Y 465.685,Z 290.08,A -85,B 0,C 180,E1 18412.714,E2 18412.714} C_VEL
LIN {X 0,Y 460.664,Z 285.135,A -85,B 0,C 180,E1 18411.156,E2 18411.156} C_VEL
LIN {X 0,Y 456.948,Z 281.577,A -85,B 0,C 180,E1 18410.033,E2 18410.033} C_VEL
LIN {X 0,Y 451.389,Z 275.772,A -85,B 0,C 180,E1 18408.374,E2 18408.374} C_VEL
LIN {X 0,Y 446.372,Z 270.545,A -85,B 0,C 180,E1 18406.908,E2 18406.908} C_VEL
LIN {X 0,Y 440.296,Z 264.388,A -85,B 0,C 180,E1 18405.208,E2 18405.208} C_VEL
LIN {X 0,Y 436.739,Z 261.019,A -85,B 0,C 180,E1 18404.289,E2 18404.289} C_VEL
LIN {X 0,Y 430.867,Z 255.082,A -85,B 0,C 180,E1 18402.84,E2 18402.84} C_VEL
LIN {X 0,Y 425.938,Z 249.955,A -85,B 0,C 180,E1 18401.677,E2 18401.677} C_VEL
LIN {X 0,Y 419.997,Z 243.778,A -85,B 0,C 180,E1 18400.358,E2 18400.358} C_VEL
LIN {X 0,Y 413.976,Z 237.17,A -85,B 0,C 180,E1 18399.08,E2 18399.08} C_VEL
LIN {X 0,Y 411.469,Z 234.417,A -85,B 0,C 180,E1 18398.558,E2 18398.558} C_VEL
LIN {X 0,Y 406.665,Z 228.522,A -85,B 0,C 180,E1 18397.529,E2 18397.529} C_VEL
LIN {X 0,Y 403.489,Z 224.079,A -85,B 0,C 180,E1 18396.804,E2 18396.804} C_VEL
LIN {X 0,Y 400.098,Z 220.235,A -85,B 0,C 180,E1 18396.032,E2 18396.032} C_VEL
LIN {X 0,Y 398.925,Z 218.088,A -85,B 0,C 180,E1 18395.733,E2 18395.733} C_VEL
LIN {X 0,Y 396.986,Z 216.669,A -85,B 0,C 180,E1 18395.296,E2 18395.296} C_VEL
LIN {X 0,Y 393.549,Z 214.33,A -85,B 0,C 180,E1 18394.498,E2 18394.498} C_VEL
LIN {X 0,Y 389.002,Z 213.152,A -85,B 0,C 180,E1 18393.339,E2 18393.339} C_VEL
LIN {X 0,Y 386.933,Z 212.985,A -85,B 0,C 180,E1 18392.503,E2 18392.503} C_VEL
LIN {X 0,Y 386.713,Z 212.977,A -85,B 0,C 180,E1 18392.17,E2 18392.17} C_VEL
LIN {X 0,Y 386.72,Z 212.898,A -85,B 0,C 180,E1 18388.408,E2 18388.408} C_VEL
LIN {X 0,Y 386.725,Z 212.975,A -85,B 0,C 180,E1 18384.437,E2 18384.437} C_VEL
LIN {X 0,Y 386.733,Z 212.973,A -85,B 0,C 180,E1 18380.587,E2 18380.587} C_VEL
LIN {X 0,Y 386.733,Z 212.965,A -85,B 0,C 180,E1 18376.678,E2 18376.678} C_VEL
LIN {X 0,Y 386.739,Z 212.964,A -85,B 0,C 180,E1 18372.847,E2 18372.847} C_VEL
LIN {X 0,Y 386.735,Z 212.978,A -85,B 0,C 180,E1 18368.774,E2 18368.774} C_VEL
LIN {X 0,Y 386.737,Z 212.995,A -85,B 0,C 180,E1 18364.894,E2 18364.894} C_VEL
LIN {X 0,Y 386.738,Z 212.973,A -85,B 0,C 180,E1 18360.889,E2 18360.889} C_VEL
LIN {X 0,Y 386.728,Z 212.961,A -85,B 0,C 180,E1 18356.887,E2 18356.887} C_VEL
LIN {X 0,Y 386.73,Z 212.964,A -85,B 0,C 180,E1 18352.871,E2 18352.871} C_VEL
LIN {X 0,Y 386.731,Z 212.987,A -85,B 0,C 180,E1 18348.97,E2 18348.97} C_VEL
LIN {X 0,Y 386.74,Z 212.993,A -85,B 0,C 180,E1 18345.016,E2 18345.016} C_VEL
LIN {X 0,Y 386.73,Z 212.981,A -85,B 0,C 180,E1 18340.987,E2 18340.987} C_VEL
LIN {X 0,Y 386.728,Z 212.976,A -85,B 0,C 180,E1 18336.972,E2 18336.972} C_VEL
LIN {X 0,Y 386.727,Z 212.909,A -85,B 0,C 180,E1 18333.098,E2 18333.098} C_VEL
LIN {X 0,Y 386.729,Z 212.945,A -85,B 0,C 180,E1 18329.123,E2 18329.123} C_VEL
LIN {X 0,Y 386.778,Z 213.287,A -85,B 0,C 180,E1 18327.591,E2 18327.591} C_VEL
LIN {X 0,Y 387.305,Z 215.102,A -85,B 0,C 180,E1 18327.17,E2 18327.17} C_VEL
LIN {X 0,Y 389.418,Z 218.046,A -85,B 0,C 180,E1 18326.58,E2 18326.58} C_VEL
LIN {X 0,Y 394.141,Z 224.076,A -85,B 0,C 180,E1 18325.371,E2 18325.371} C_VEL
LIN {X 0,Y 398.328,Z 229.854,A -85,B 0,C 180,E1 18324.338,E2 18324.338} C_VEL
LIN {X 0,Y 407.059,Z 242.391,A -85,B 0,C 180,E1 18322.314,E2 18322.314} C_VEL
LIN {X 0,Y 417.47,Z 258.432,A -85,B 0,C 180,E1 18320.089,E2 18320.089} C_VEL
LIN {X 0,Y 428.191,Z 276.706,A -85,B 0,C 180,E1 18317.963,E2 18317.963} C_VEL
LIN {X 0,Y 438.149,Z 295.19,A -85,B 0,C 180,E1 18316.117,E2 18316.117} C_VEL
LIN {X 0,Y 444.86,Z 309.097,A -85,B 0,C 180,E1 18314.92,E2 18314.92} C_VEL
LIN {X 0,Y 435.224,Z 520.537,A -85,B 0,C 180,E1 18311.419,E2 18311.419} C_VEL
LIN {X 0,Y 433.675,Z 538.855,A -85,B 0,C 180,E1 18310.996,E2 18310.996} C_VEL
LIN {X 0,Y 431.127,Z 560.478,A -85,B 0,C 180,E1 18310.314,E2 18310.314} C_VEL
LIN {X 0,Y 427.788,Z 581.877,A -85,B 0,C 180,E1 18309.383,E2 18309.383} C_VEL
LIN {X 0,Y 424.59,Z 599.374,A -85,B 0,C 180,E1 18308.435,E2 18308.435} C_VEL
LIN {X 0,Y 421.315,Z 615.239,A -85,B 0,C 180,E1 18307.407,E2 18307.407} C_VEL
LIN {X 0,Y 417.813,Z 630.684,A -85,B 0,C 180,E1 18306.23,E2 18306.23} C_VEL
LIN {X 0,Y 414.12,Z 645.668,A -85,B 0,C 180,E1 18304.901,E2 18304.901} C_VEL
LIN {X 0,Y 410.013,Z 661.403,A -85,B 0,C 180,E1 18303.273,E2 18303.273} C_VEL
LIN {X 0,Y 404.982,Z 679.447,A -85,B 0,C 180,E1 18301.048,E2 18301.048} C_VEL
LIN {X 0,Y 401.103,Z 692.871,A -85,B 0,C 180,E1 18299.081,E2 18299.081} C_VEL
LIN {X 0,Y 397.647,Z 704.762,A -85,B 0,C 180,E1 18297.069,E2 18297.069} C_VEL
LIN {X 0,Y 394.62,Z 715.259,A -85,B 0,C 180,E1 18295.03,E2 18295.03} C_VEL
LIN {X 0,Y 391.849,Z 725.151,A -85,B 0,C 180,E1 18292.818,E2 18292.818} C_VEL
LIN {X 0,Y 389.425,Z 734.335,A -85,B 0,C 180,E1 18290.435,E2 18290.435} C_VEL
LIN {X 0,Y 387.217,Z 743.652,A -85,B 0,C 180,E1 18287.583,E2 18287.583} C_VEL
LIN {X 0,Y 385.463,Z 752.298,A -85,B 0,C 180,E1 18284.264,E2 18284.264} C_VEL
LIN {X 0,Y 384.601,Z 757.909,A -85,B 0,C 180,E1 18281.546,E2 18281.546} C_VEL
LIN {X 0,Y 384.148,Z 762.074,A -85,B 0,C 180,E1 18278.984,E2 18278.984} C_VEL
LIN {X 0,Y 383.976,Z 765.171,A -85,B 0,C 180,E1 18276.428,E2 18276.428} C_VEL
LIN {X 0,Y 383.94,Z 767.23,A -85,B 0,C 180,E1 18273.882,E2 18273.882} C_VEL
LIN {X 0,Y 383.952,Z 768.24,A -85,B 0,C 180,E1 18271.492,E2 18271.492} C_VEL
LIN {X 0,Y 383.959,Z 768.358,A -85,B 0,C 180,E1 18269.105,E2 18269.105} C_VEL
LIN {X 0,Y 383.938,Z 767.496,A -85,B 0,C 180,E1 18266.566,E2 18266.566} C_VEL
LIN {X 0,Y 383.96,Z 765.615,A -85,B 0,C 180,E1 18264.022,E2 18264.022} C_VEL
LIN {X 0,Y 384.109,Z 762.7,A -85,B 0,C 180,E1 18261.468,E2 18261.468} C_VEL
LIN {X 0,Y 384.498,Z 758.72,A -85,B 0,C 180,E1 18258.906,E2 18258.906} C_VEL
LIN {X 0,Y 385.229,Z 753.634,A -85,B 0,C 180,E1 18256.34,E2 18256.34} C_VEL
LIN {X 0,Y 386.311,Z 747.785,A -85,B 0,C 180,E1 18253.924,E2 18253.924} C_VEL
LIN {X 0,Y 387.835,Z 740.839,A -85,B 0,C 180,E1 18251.514,E2 18251.514} C_VEL
LIN {X 0,Y 389.84,Z 732.71,A -85,B 0,C 180,E1 18249.117,E2 18249.117} C_VEL
LIN {X 0,Y 392.547,Z 722.675,A -85,B 0,C 180,E1 18246.59,E2 18246.59} C_VEL
LIN {X 0,Y 396.519,Z 708.72,A -85,B 0,C 180,E1 18243.656,E2 18243.656} C_VEL
LIN {X 0,Y 400.075,Z 696.432,A -85,B 0,C 180,E1 18241.491,E2 18241.491} C_VEL
LIN {X 0,Y 403.705,Z 683.865,A -85,B 0,C 180,E1 18239.573,E2 18239.573} C_VEL
LIN {X 0,Y 407.314,Z 671.113,A -85,B 0,C 180,E1 18237.879,E2 18237.879} C_VEL
LIN {X 0,Y 411.049,Z 657.447,A -85,B 0,C 180,E1 18236.298,E2 18236.298} C_VEL
LIN {X 0,Y 414.833,Z 642.823,A -85,B 0,C 180,E1 18234.831,E2 18234.831} C_VEL
LIN {X 0,Y 418.739,Z 626.764,A -85,B 0,C 180,E1 18233.45,E2 18233.45} C_VEL
LIN {X 0,Y 423.348,Z 605.747,A -85,B 0,C 180,E1 18231.949,E2 18231.949} C_VEL
LIN {X 0,Y 426.922,Z 586.851,A -85,B 0,C 180,E1 18230.868,E2 18230.868} C_VEL
LIN {X 0,Y 429.644,Z 570.215,A -85,B 0,C 180,E1 18230.085,E2 18230.085} C_VEL
LIN {X 0,Y 432.057,Z 552.822,A -85,B 0,C 180,E1 18229.426,E2 18229.426} C_VEL
LIN {X 0,Y 434.021,Z 535.314,A -85,B 0,C 180,E1 18228.913,E2 18228.913} C_VEL
LIN {X 0,Y 435.447,Z 516.941,A -85,B 0,C 180,E1 18228.511,E2 18228.511} C_VEL
LIN {X 0,Y 444.782,Z 308.67,A -85,B 0,C 180,E1 18225.061,E2 18225.061} C_VEL
LIN {X 0,Y 434.463,Z 288.089,A -85,B 0,C 180,E1 18223.211,E2 18223.211} C_VEL
LIN {X 0,Y 423.747,Z 268.892,A -85,B 0,C 180,E1 18221.174,E2 18221.174} C_VEL
LIN {X 0,Y 413.03,Z 251.472,A -85,B 0,C 180,E1 18218.986,E2 18218.986} C_VEL
LIN {X 0,Y 402.814,Z 236.087,A -85,B 0,C 180,E1 18216.719,E2 18216.719} C_VEL
LIN {X 0,Y 396.288,Z 226.993,A -85,B 0,C 180,E1 18215.163,E2 18215.163} C_VEL
LIN {X 0,Y 389.8,Z 218.374,A -85,B 0,C 180,E1 18213.515,E2 18213.515} C_VEL
LIN {X 0,Y 387.452,Z 215.437,A -85,B 0,C 180,E1 18212.882,E2 18212.882} C_VEL
LIN {X 0,Y 386.804,Z 213.421,A -85,B 0,C 180,E1 18212.462,E2 18212.462} C_VEL
LIN {X 0,Y 386.701,Z 212.972,A -85,B 0,C 180,E1 18211.443,E2 18211.443} C_VEL
LIN {X 0,Y 386.694,Z 212.904,A -85,B 0,C 180,E1 18207.528,E2 18207.528} C_VEL
LIN {X 0,Y 386.7,Z 212.99,A -85,B 0,C 180,E1 18203.627,E2 18203.627} C_VEL
LIN {X 0,Y 386.701,Z 212.997,A -85,B 0,C 180,E1 18199.642,E2 18199.642} C_VEL
LIN {X 0,Y 386.702,Z 212.994,A -85,B 0,C 180,E1 18195.6,E2 18195.6} C_VEL
LIN {X 0,Y 386.702,Z 212.976,A -85,B 0,C 180,E1 18191.636,E2 18191.636} C_VEL
LIN {X 0,Y 386.697,Z 212.966,A -85,B 0,C 180,E1 18187.727,E2 18187.727} C_VEL
LIN {X 0,Y 386.697,Z 212.974,A -85,B 0,C 180,E1 18183.855,E2 18183.855} C_VEL
LIN {X 0,Y 386.698,Z 212.996,A -85,B 0,C 180,E1 18179.852,E2 18179.852} C_VEL
LIN {X 0,Y 386.699,Z 212.994,A -85,B 0,C 180,E1 18175.848,E2 18175.848} C_VEL
LIN {X 0,Y 386.697,Z 212.973,A -85,B 0,C 180,E1 18171.97,E2 18171.97} C_VEL
LIN {X 0,Y 386.698,Z 212.969,A -85,B 0,C 180,E1 18168.062,E2 18168.062} C_VEL
LIN {X 0,Y 386.696,Z 212.979,A -85,B 0,C 180,E1 18164.092,E2 18164.092} C_VEL
LIN {X 0,Y 386.701,Z 212.989,A -85,B 0,C 180,E1 18160.043,E2 18160.043} C_VEL
LIN {X 0,Y 386.703,Z 212.998,A -85,B 0,C 180,E1 18156.049,E2 18156.049} C_VEL
LIN {X 0,Y 386.693,Z 212.899,A -85,B 0,C 180,E1 18152.094,E2 18152.094} C_VEL
LIN {X 0,Y 386.702,Z 212.994,A -85,B 0,C 180,E1 18148.165,E2 18148.165} C_VEL
LIN {X 0,Y 386.763,Z 213.145,A -85,B 0,C 180,E1 18147.294,E2 18147.294} C_VEL
LIN {X 0,Y 387.075,Z 214.528,A -85,B 0,C 180,E1 18146.927,E2 18146.927} C_VEL
LIN {X 0,Y 388.94,Z 217.566,A -85,B 0,C 180,E1 18146.395,E2 18146.395} C_VEL
LIN {X 0,Y 391.479,Z 219.714,A -85,B 0,C 180,E1 18145.768,E2 18145.768} C_VEL
LIN {X 0,Y 393.924,Z 223.469,A -85,B 0,C 180,E1 18145.128,E2 18145.128} C_VEL
LIN {X 0,Y 396.138,Z 225.687,A -85,B 0,C 180,E1 18144.6,E2 18144.6} C_VEL
LIN {X 0,Y 399.354,Z 229.954,A -85,B 0,C 180,E1 18143.824,E2 18143.824} C_VEL
LIN {X 0,Y 408.755,Z 241.707,A -85,B 0,C 180,E1 18141.72,E2 18141.72} C_VEL
LIN {X 0,Y 415.184,Z 248.738,A -85,B 0,C 180,E1 18140.387,E2 18140.387} C_VEL
LIN {X 0,Y 421.546,Z 255.43,A -85,B 0,C 180,E1 18139.016,E2 18139.016} C_VEL
LIN {X 0,Y 428.307,Z 262.278,A -85,B 0,C 180,E1 18137.48,E2 18137.48} C_VEL
LIN {X 0,Y 435.461,Z 269.272,A -85,B 0,C 180,E1 18135.73,E2 18135.73} C_VEL
LIN {X 0,Y 442.466,Z 276.229,A -85,B 0,C 180,E1 18133.873,E2 18133.873} C_VEL
LIN {X 0,Y 449.445,Z 283.306,A -85,B 0,C 180,E1 18131.861,E2 18131.861} C_VEL
LIN {X 0,Y 456.316,Z 290.253,A -85,B 0,C 180,E1 18129.823,E2 18129.823} C_VEL
LIN {X 0,Y 463.53,Z 297.377,A -85,B 0,C 180,E1 18127.617,E2 18127.617} C_VEL
LIN {X 0,Y 466.859,Z 300.775,A -85,B 0,C 180,E1 18126.567,E2 18126.567} C_VEL
LIN {X 0,Y 472.149,Z 305.526,A -85,B 0,C 180,E1 18124.87,E2 18124.87} C_VEL
LIN {X 0,Y 477.756,Z 311.248,A -85,B 0,C 180,E1 18122.962,E2 18122.962} C_VEL
LIN {X 0,Y 481.158,Z 314.204,A -85,B 0,C 180,E1 18121.794,E2 18121.794} C_VEL
LIN {X 0,Y 486.327,Z 319.197,A -85,B 0,C 180,E1 18119.926,E2 18119.926} C_VEL
LIN {X 0,Y 489.149,Z 321.666,A -85,B 0,C 180,E1 18118.875,E2 18118.875} C_VEL
LIN {X 0,Y 493.879,Z 326.293,A -85,B 0,C 180,E1 18117.024,E2 18117.024} C_VEL
LIN {X 0,Y 497.304,Z 328.979,A -85,B 0,C 180,E1 18115.643,E2 18115.643} C_VEL
LIN {X 0,Y 501.797,Z 333.501,A -85,B 0,C 180,E1 18113.669,E2 18113.669} C_VEL
LIN {X 0,Y 505.968,Z 336.698,A -85,B 0,C 180,E1 18111.749,E2 18111.749} C_VEL
LIN {X 0,Y 509.975,Z 340.844,A -85,B 0,C 180,E1 18109.706,E2 18109.706} C_VEL
LIN {X 0,Y 513.925,Z 343.512,A -85,B 0,C 180,E1 18107.549,E2 18107.549} C_VEL
LIN {X 0,Y 515.239,Z 344.835,A -85,B 0,C 180,E1 18106.747,E2 18106.747} C_VEL
LIN {X 0,Y 518.403,Z 348.267,A -85,B 0,C 180,E1 18104.634,E2 18104.634} C_VEL
LIN {X 0,Y 521.379,Z 350.433,A -85,B 0,C 180,E1 18102.402,E2 18102.402} C_VEL
LIN {X 0,Y 524.276,Z 351.911,A -85,B 0,C 180,E1 18099.882,E2 18099.882} C_VEL
LIN {X 0,Y 525.938,Z 354.384,A -85,B 0,C 180,E1 18097.866,E2 18097.866} C_VEL
LIN {X 0,Y 527.436,Z 356.057,A -85,B 0,C 180,E1 18095.547,E2 18095.547} C_VEL
LIN {X 0,Y 528.561,Z 357.041,A -85,B 0,C 180,E1 18092.927,E2 18092.927} C_VEL
LIN {X 0,Y 528.964,Z 357.306,A -85,B 0,C 180,E1 18090.433,E2 18090.433} C_VEL
LIN {X 0,Y 528.754,Z 357.122,A -85,B 0,C 180,E1 18087.833,E2 18087.833} C_VEL
LIN {X 0,Y 527.876,Z 356.447,A -85,B 0,C 180,E1 18085.329,E2 18085.329} C_VEL
LIN {X 0,Y 526.416,Z 354.923,A -85,B 0,C 180,E1 18082.799,E2 18082.799} C_VEL
LIN {X 0,Y 524.768,Z 352.767,A -85,B 0,C 180,E1 18080.681,E2 18080.681} C_VEL
LIN {X 0,Y 523.732,Z 351.506,A -85,B 0,C 180,E1 18079.552,E2 18079.552} C_VEL
LIN {X 0,Y 520.88,Z 350.118,A -85,B 0,C 180,E1 18077.205,E2 18077.205} C_VEL
LIN {X 0,Y 517.759,Z 347.676,A -85,B 0,C 180,E1 18074.928,E2 18074.928} C_VEL
LIN {X 0,Y 514.786,Z 344.176,A -85,B 0,C 180,E1 18072.947,E2 18072.947} C_VEL
LIN {X 0,Y 510.204,Z 341.043,A -85,B 0,C 180,E1 18070.423,E2 18070.423} C_VEL
LIN {X 0,Y 506.113,Z 336.869,A -85,B 0,C 180,E1 18068.322,E2 18068.322} C_VEL
LIN {X 0,Y 504.155,Z 335.204,A -85,B 0,C 180,E1 18067.374,E2 18067.374} C_VEL
LIN {X 0,Y 499.528,Z 331.455,A -85,B 0,C 180,E1 18065.335,E2 18065.335} C_VEL
LIN {X 0,Y 495.953,Z 327.778,A -85,B 0,C 180,E1 18063.803,E2 18063.803} C_VEL
LIN {X 0,Y 491.145,Z 323.804,A -85,B 0,C 180,E1 18061.89,E2 18061.89} C_VEL
LIN {X 0,Y 487.381,Z 319.974,A -85,B 0,C 180,E1 18060.443,E2 18060.443} C_VEL
LIN {X 0,Y 481.972,Z 315.118,A -85,B 0,C 180,E1 18058.502,E2 18058.502} C_VEL
LIN {X 0,Y 479.317,Z 312.467,A -85,B 0,C 180,E1 18057.557,E2 18057.557} C_VEL
LIN {X 0,Y 474.035,Z 307.653,A -85,B 0,C 180,E1 18055.777,E2 18055.777} C_VEL
LIN {X 0,Y 471.325,Z 304.916,A -85,B 0,C 180,E1 18054.867,E2 18054.867} C_VEL
LIN {X 0,Y 466.12,Z 299.962,A -85,B 0,C 180,E1 18053.2,E2 18053.2} C_VEL
LIN {X 0,Y 463.229,Z 297.124,A -85,B 0,C 180,E1 18052.289,E2 18052.289} C_VEL
LIN {X 0,Y 457.753,Z 291.465,A -85,B 0,C 180,E1 18050.593,E2 18050.593} C_VEL
LIN {X 0,Y 451.856,Z 285.783,A -85,B 0,C 180,E1 18048.844,E2 18048.844} C_VEL
LIN {X 0,Y 448.512,Z 282.468,A -85,B 0,C 180,E1 18047.86,E2 18047.86} C_VEL
LIN {X 0,Y 441.888,Z 275.732,A -85,B 0,C 180,E1 18045.972,E2 18045.972} C_VEL
LIN {X 0,Y 435.137,Z 268.998,A -85,B 0,C 180,E1 18044.188,E2 18044.188} C_VEL
LIN {X 0,Y 429.868,Z 263.635,A -85,B 0,C 180,E1 18042.895,E2 18042.895} C_VEL
LIN {X 0,Y 424.037,Z 258.106,A -85,B 0,C 180,E1 18041.544,E2 18041.544} C_VEL
LIN {X 0,Y 416.558,Z 250.203,A -85,B 0,C 180,E1 18039.904,E2 18039.904} C_VEL
LIN {X 0,Y 410.435,Z 243.568,A -85,B 0,C 180,E1 18038.629,E2 18038.629} C_VEL
LIN {X 0,Y 404.857,Z 236.974,A -85,B 0,C 180,E1 18037.435,E2 18037.435} C_VEL
LIN {X 0,Y 400.219,Z 230.889,A -85,B 0,C 180,E1 18036.374,E2 18036.374} C_VEL
LIN {X 0,Y 396.383,Z 226.124,A -85,B 0,C 180,E1 18035.464,E2 18035.464} C_VEL
LIN {X 0,Y 395.234,Z 224.653,A -85,B 0,C 180,E1 18035.182,E2 18035.182} C_VEL
LIN {X 0,Y 392.3,Z 221.317,A -85,B 0,C 180,E1 18034.46,E2 18034.46} C_VEL
LIN {X 0,Y 391.119,Z 219.131,A -85,B 0,C 180,E1 18034.135,E2 18034.135} C_VEL
LIN {X 0,Y 388.185,Z 216.684,A -85,B 0,C 180,E1 18033.407,E2 18033.407} C_VEL
LIN {X 0,Y 386.861,Z 213.743,A -85,B 0,C 180,E1 18032.934,E2 18032.934} C_VEL
LIN {X 0,Y 386.74,Z 213.002,A -85,B 0,C 180,E1 18032.532,E2 18032.532} C_VEL
LIN {X 0,Y 386.713,Z 212.977,A -85,B 0,C 180,E1 18032.17,E2 18032.17} C_VEL
LIN {X 0,Y 385.675,Z 213.126,A -85,B 0,C 180,E1 18031.029,E2 18031.029} C_VEL
LIN {X 0,Y 379.173,Z 213.839,A -85,B 0,C 180,E1 18027.724,E2 18027.724} C_VEL
LIN {X 0,Y 378.779,Z 213.886,A -85,B 0,C 180,E1 18026.966,E2 18026.966} C_VEL
LIN {X 0,Y 378.798,Z 213.97,A -85,B 0,C 180,E1 18022.912,E2 18022.912} C_VEL
LIN {X 0,Y 378.802,Z 213.976,A -85,B 0,C 180,E1 18018.786,E2 18018.786} C_VEL
LIN {X 0,Y 378.8,Z 213.982,A -85,B 0,C 180,E1 18014.679,E2 18014.679} C_VEL
LIN {X 0,Y 378.788,Z 213.968,A -85,B 0,C 180,E1 18010.648,E2 18010.648} C_VEL
LIN {X 0,Y 378.786,Z 213.954,A -85,B 0,C 180,E1 18006.67,E2 18006.67} C_VEL
LIN {X 0,Y 378.784,Z 213.953,A -85,B 0,C 180,E1 18002.723,E2 18002.723} C_VEL
LIN {X 0,Y 378.791,Z 213.971,A -85,B 0,C 180,E1 17998.79,E2 17998.79} C_VEL
LIN {X 0,Y 378.781,Z 213.983,A -85,B 0,C 180,E1 17994.699,E2 17994.699} C_VEL
LIN {X 0,Y 378.781,Z 213.961,A -85,B 0,C 180,E1 17990.733,E2 17990.733} C_VEL
LIN {X 0,Y 378.776,Z 213.955,A -85,B 0,C 180,E1 17986.723,E2 17986.723} C_VEL
LIN {X 0,Y 378.779,Z 213.957,A -85,B 0,C 180,E1 17982.803,E2 17982.803} C_VEL
LIN {X 0,Y 378.777,Z 213.964,A -85,B 0,C 180,E1 17978.798,E2 17978.798} C_VEL
LIN {X 0,Y 378.778,Z 213.953,A -85,B 0,C 180,E1 17974.849,E2 17974.849} C_VEL
LIN {X 0,Y 378.768,Z 213.89,A -85,B 0,C 180,E1 17970.888,E2 17970.888} C_VEL
LIN {X 0,Y 378.867,Z 214.315,A -85,B 0,C 180,E1 17969.379,E2 17969.379} C_VEL
LIN {X 0,Y 379.387,Z 216.152,A -85,B 0,C 180,E1 17969.008,E2 17969.008} C_VEL
LIN {X 0,Y 381.487,Z 219.049,A -85,B 0,C 180,E1 17968.385,E2 17968.385} C_VEL
LIN {X 0,Y 383.633,Z 220.739,A -85,B 0,C 180,E1 17967.813,E2 17967.813} C_VEL
LIN {X 0,Y 386.139,Z 224.573,A -85,B 0,C 180,E1 17967.102,E2 17967.102} C_VEL
LIN {X 0,Y 390.199,Z 229.482,A -85,B 0,C 180,E1 17966.039,E2 17966.039} C_VEL
LIN {X 0,Y 399.952,Z 243.372,A -85,B 0,C 180,E1 17963.616,E2 17963.616} C_VEL
LIN {X 0,Y 410.456,Z 259.462,A -85,B 0,C 180,E1 17961.239,E2 17961.239} C_VEL
LIN {X 0,Y 420.584,Z 276.384,A -85,B 0,C 180,E1 17959.127,E2 17959.127} C_VEL
LIN {X 0,Y 431.129,Z 295.675,A -85,B 0,C 180,E1 17957.079,E2 17957.079} C_VEL
LIN {X 0,Y 439.072,Z 311.889,A -85,B 0,C 180,E1 17955.61,E2 17955.61} C_VEL
LIN {X 0,Y 429.244,Z 520.362,A -85,B 0,C 180,E1 17952.127,E2 17952.127} C_VEL
LIN {X 0,Y 427.653,Z 538.68,A -85,B 0,C 180,E1 17951.701,E2 17951.701} C_VEL
LIN {X 0,Y 425.031,Z 560.302,A -85,B 0,C 180,E1 17951.015,E2 17951.015} C_VEL
LIN {X 0,Y 421.595,Z 581.701,A -85,B 0,C 180,E1 17950.077,E2 17950.077} C_VEL
LIN {X 0,Y 418.303,Z 599.197,A -85,B 0,C 180,E1 17949.121,E2 17949.121} C_VEL
LIN {X 0,Y 414.923,Z 615.062,A -85,B 0,C 180,E1 17948.085,E2 17948.085} C_VEL
LIN {X 0,Y 411.308,Z 630.507,A -85,B 0,C 180,E1 17946.897,E2 17946.897} C_VEL
LIN {X 0,Y 407.491,Z 645.49,A -85,B 0,C 180,E1 17945.554,E2 17945.554} C_VEL
LIN {X 0,Y 403.239,Z 661.225,A -85,B 0,C 180,E1 17943.907,E2 17943.907} C_VEL
LIN {X 0,Y 397.841,Z 679.86,A -85,B 0,C 180,E1 17941.569,E2 17941.569} C_VEL
LIN {X 0,Y 393.988,Z 692.693,A -85,B 0,C 180,E1 17939.658,E2 17939.658} C_VEL
LIN {X 0,Y 390.384,Z 704.583,A -85,B 0,C 180,E1 17937.615,E2 17937.615} C_VEL
LIN {X 0,Y 387.225,Z 715.08,A -85,B 0,C 180,E1 17935.542,E2 17935.542} C_VEL
LIN {X 0,Y 384.324,Z 724.972,A -85,B 0,C 180,E1 17933.291,E2 17933.291} C_VEL
LIN {X 0,Y 381.775,Z 734.156,A -85,B 0,C 180,E1 17930.863,E2 17930.863} C_VEL
LIN {X 0,Y 379.442,Z 743.474,A -85,B 0,C 180,E1 17927.955,E2 17927.955} C_VEL
LIN {X 0,Y 377.58,Z 752.12,A -85,B 0,C 180,E1 17924.569,E2 17924.569} C_VEL
LIN {X 0,Y 376.657,Z 757.731,A -85,B 0,C 180,E1 17921.793,E2 17921.793} C_VEL
LIN {X 0,Y 376.17,Z 761.897,A -85,B 0,C 180,E1 17919.176,E2 17919.176} C_VEL
LIN {X 0,Y 375.978,Z 764.995,A -85,B 0,C 180,E1 17916.566,E2 17916.566} C_VEL
LIN {X 0,Y 375.941,Z 767.055,A -85,B 0,C 180,E1 17913.965,E2 17913.965} C_VEL
LIN {X 0,Y 375.955,Z 768.065,A -85,B 0,C 180,E1 17911.524,E2 17911.524} C_VEL
LIN {X 0,Y 375.96,Z 768.183,A -85,B 0,C 180,E1 17909.086,E2 17909.086} C_VEL
LIN {X 0,Y 375.94,Z 767.321,A -85,B 0,C 180,E1 17906.493,E2 17906.493} C_VEL
LIN {X 0,Y 375.966,Z 765.44,A -85,B 0,C 180,E1 17903.894,E2 17903.894} C_VEL
LIN {X 0,Y 376.127,Z 762.523,A -85,B 0,C 180,E1 17901.286,E2 17901.286} C_VEL
LIN {X 0,Y 376.548,Z 758.542,A -85,B 0,C 180,E1 17898.669,E2 17898.669} C_VEL
LIN {X 0,Y 377.332,Z 753.456,A -85,B 0,C 180,E1 17896.048,E2 17896.048} C_VEL
LIN {X 0,Y 378.569,Z 747.207,A -85,B 0,C 180,E1 17893.428,E2 17893.428} C_VEL
LIN {X 0,Y 380.214,Z 740.192,A -85,B 0,C 180,E1 17890.971,E2 17890.971} C_VEL
LIN {X 0,Y 382.516,Z 731.448,A -85,B 0,C 180,E1 17888.376,E2 17888.376} C_VEL
LIN {X 0,Y 386.01,Z 719.29,A -85,B 0,C 180,E1 17885.356,E2 17885.356} C_VEL
LIN {X 0,Y 389.674,Z 706.958,A -85,B 0,C 180,E1 17882.827,E2 17882.827} C_VEL
LIN {X 0,Y 393.18,Z 695.363,A -85,B 0,C 180,E1 17880.777,E2 17880.777} C_VEL
LIN {X 0,Y 396.985,Z 682.688,A -85,B 0,C 180,E1 17878.834,E2 17878.834} C_VEL
LIN {X 0,Y 400.723,Z 669.957,A -85,B 0,C 180,E1 17877.137,E2 17877.137} C_VEL
LIN {X 0,Y 404.613,Z 656.182,A -85,B 0,C 180,E1 17875.54,E2 17875.54} C_VEL
LIN {X 0,Y 408.799,Z 640.513,A -85,B 0,C 180,E1 17873.973,E2 17873.973} C_VEL
LIN {X 0,Y 413.911,Z 619.664,A -85,B 0,C 180,E1 17872.244,E2 17872.244} C_VEL
LIN {X 0,Y 417.659,Z 602.384,A -85,B 0,C 180,E1 17871.072,E2 17871.072} C_VEL
LIN {X 0,Y 420.928,Z 585.431,A -85,B 0,C 180,E1 17870.113,E2 17870.113} C_VEL
LIN {X 0,Y 423.626,Z 569.296,A -85,B 0,C 180,E1 17869.356,E2 17869.356} C_VEL
LIN {X 0,Y 426.064,Z 552.109,A -85,B 0,C 180,E1 17868.706,E2 17868.706} C_VEL
LIN {X 0,Y 428.075,Z 534.507,A -85,B 0,C 180,E1 17868.191,E2 17868.191} C_VEL
LIN {X 0,Y 429.584,Z 515.021,A -85,B 0,C 180,E1 17867.768,E2 17867.768} C_VEL
LIN {X 0,Y 438.97,Z 311.613,A -85,B 0,C 180,E1 17864.37,E2 17864.37} C_VEL
LIN {X 0,Y 429.453,Z 292.558,A -85,B 0,C 180,E1 17862.606,E2 17862.606} C_VEL
LIN {X 0,Y 419.385,Z 274.321,A -85,B 0,C 180,E1 17860.631,E2 17860.631} C_VEL
LIN {X 0,Y 409.093,Z 257.359,A -85,B 0,C 180,E1 17858.466,E2 17858.466} C_VEL
LIN {X 0,Y 398.132,Z 240.663,A -85,B 0,C 180,E1 17855.948,E2 17855.948} C_VEL
LIN {X 0,Y 392.406,Z 232.784,A -85,B 0,C 180,E1 17854.538,E2 17854.538} C_VEL
LIN {X 0,Y 387.01,Z 225.414,A -85,B 0,C 180,E1 17853.123,E2 17853.123} C_VEL
LIN {X 0,Y 384.188,Z 221.841,A -85,B 0,C 180,E1 17852.355,E2 17852.355} C_VEL
LIN {X 0,Y 383.218,Z 220.232,A -85,B 0,C 180,E1 17852.071,E2 17852.071} C_VEL
LIN {X 0,Y 380.311,Z 217.773,A -85,B 0,C 180,E1 17851.283,E2 17851.283} C_VEL
LIN {X 0,Y 378.901,Z 214.531,A -85,B 0,C 180,E1 17850.697,E2 17850.697} C_VEL
LIN {X 0,Y 378.763,Z 213.93,A -85,B 0,C 180,E1 17850.03,E2 17850.03} C_VEL
LIN {X 0,Y 378.767,Z 213.917,A -85,B 0,C 180,E1 17846.159,E2 17846.159} C_VEL
LIN {X 0,Y 378.78,Z 213.957,A -85,B 0,C 180,E1 17842.342,E2 17842.342} C_VEL
LIN {X 0,Y 378.786,Z 213.957,A -85,B 0,C 180,E1 17838.468,E2 17838.468} C_VEL
LIN {X 0,Y 378.786,Z 213.969,A -85,B 0,C 180,E1 17834.523,E2 17834.523} C_VEL
LIN {X 0,Y 378.781,Z 213.984,A -85,B 0,C 180,E1 17830.495,E2 17830.495} C_VEL
LIN {X 0,Y 378.777,Z 213.967,A -85,B 0,C 180,E1 17826.518,E2 17826.518} C_VEL
LIN {X 0,Y 378.777,Z 213.954,A -85,B 0,C 180,E1 17822.572,E2 17822.572} C_VEL
LIN {X 0,Y 378.779,Z 213.957,A -85,B 0,C 180,E1 17818.639,E2 17818.639} C_VEL
LIN {X 0,Y 378.781,Z 213.98,A -85,B 0,C 180,E1 17814.699,E2 17814.699} C_VEL
LIN {X 0,Y 378.784,Z 213.981,A -85,B 0,C 180,E1 17810.734,E2 17810.734} C_VEL
LIN {X 0,Y 378.776,Z 213.963,A -85,B 0,C 180,E1 17806.723,E2 17806.723} C_VEL
LIN {X 0,Y 378.779,Z 213.957,A -85,B 0,C 180,E1 17802.803,E2 17802.803} C_VEL
LIN {X 0,Y 378.776,Z 213.959,A -85,B 0,C 180,E1 17798.798,E2 17798.798} C_VEL
LIN {X 0,Y 378.775,Z 213.932,A -85,B 0,C 180,E1 17794.849,E2 17794.849} C_VEL
LIN {X 0,Y 378.769,Z 213.896,A -85,B 0,C 180,E1 17790.888,E2 17790.888} C_VEL
LIN {X 0,Y 378.819,Z 214.103,A -85,B 0,C 180,E1 17789.199,E2 17789.199} C_VEL
LIN {X 0,Y 379.146,Z 215.591,A -85,B 0,C 180,E1 17788.787,E2 17788.787} C_VEL
LIN {X 0,Y 380.892,Z 218.499,A -85,B 0,C 180,E1 17788.242,E2 17788.242} C_VEL
LIN {X 0,Y 383.642,Z 220.692,A -85,B 0,C 180,E1 17787.505,E2 17787.505} C_VEL
LIN {X 0,Y 386.024,Z 224.434,A -85,B 0,C 180,E1 17786.826,E2 17786.826} C_VEL
LIN {X 0,Y 388.461,Z 226.784,A -85,B 0,C 180,E1 17786.2,E2 17786.2} C_VEL
LIN {X 0,Y 391.603,Z 231.002,A -85,B 0,C 180,E1 17785.381,E2 17785.381} C_VEL
LIN {X 0,Y 393.256,Z 232.942,A -85,B 0,C 180,E1 17784.971,E2 17784.971} C_VEL
LIN {X 0,Y 398.125,Z 239.388,A -85,B 0,C 180,E1 17783.784,E2 17783.784} C_VEL
LIN {X 0,Y 405.911,Z 248.857,A -85,B 0,C 180,E1 17782.032,E2 17782.032} C_VEL
LIN {X 0,Y 412.059,Z 255.64,A -85,B 0,C 180,E1 17780.748,E2 17780.748} C_VEL
LIN {X 0,Y 418.671,Z 262.483,A -85,B 0,C 180,E1 17779.353,E2 17779.353} C_VEL
LIN {X 0,Y 425.532,Z 269.359,A -85,B 0,C 180,E1 17777.822,E2 17777.822} C_VEL
LIN {X 0,Y 433.447,Z 276.883,A -85,B 0,C 180,E1 17775.932,E2 17775.932} C_VEL
LIN {X 0,Y 440.308,Z 283.645,A -85,B 0,C 180,E1 17774.143,E2 17774.143} C_VEL
LIN {X 0,Y 447.261,Z 290.622,A -85,B 0,C 180,E1 17772.175,E2 17772.175} C_VEL
LIN {X 0,Y 454.472,Z 297.855,A -85,B 0,C 180,E1 17770.036,E2 17770.036} C_VEL
LIN {X 0,Y 461.646,Z 304.899,A -85,B 0,C 180,E1 17767.863,E2 17767.863} C_VEL
LIN {X 0,Y 468.703,Z 311.851,A -85,B 0,C 180,E1 17765.613,E2 17765.613} C_VEL
LIN {X 0,Y 471.654,Z 314.548,A -85,B 0,C 180,E1 17764.659,E2 17764.659} C_VEL
LIN {X 0,Y 476.915,Z 319.56,A -85,B 0,C 180,E1 17762.884,E2 17762.884} C_VEL
LIN {X 0,Y 479.838,Z 322.23,A -85,B 0,C 180,E1 17761.88,E2 17761.88} C_VEL
LIN {X 0,Y 485.012,Z 327.085,A -85,B 0,C 180,E1 17760.018,E2 17760.018} C_VEL
LIN {X 0,Y 487.572,Z 329.335,A -85,B 0,C 180,E1 17759.076,E2 17759.076} C_VEL
LIN {X 0,Y 492.389,Z 334.013,A -85,B 0,C 180,E1 17757.196,E2 17757.196} C_VEL
LIN {X 0,Y 495.913,Z 336.808,A -85,B 0,C 180,E1 17755.782,E2 17755.782} C_VEL
LIN {X 0,Y 500.497,Z 341.32,A -85,B 0,C 180,E1 17753.795,E2 17753.795} C_VEL
LIN {X 0,Y 504.612,Z 344.468,A -85,B 0,C 180,E1 17751.907,E2 17751.907} C_VEL
LIN {X 0,Y 508.889,Z 348.796,A -85,B 0,C 180,E1 17749.749,E2 17749.749} C_VEL
LIN {X 0,Y 512.884,Z 351.449,A -85,B 0,C 180,E1 17747.573,E2 17747.573} C_VEL
LIN {X 0,Y 516.654,Z 355.583,A -85,B 0,C 180,E1 17745.143,E2 17745.143} C_VEL
LIN {X 0,Y 519.769,Z 357.999,A -85,B 0,C 180,E1 17742.892,E2 17742.892} C_VEL
LIN {X 0,Y 522.581,Z 359.389,A -85,B 0,C 180,E1 17740.583,E2 17740.583} C_VEL
LIN {X 0,Y 523.57,Z 360.437,A -85,B 0,C 180,E1 17739.563,E2 17739.563} C_VEL
LIN {X 0,Y 525.276,Z 362.684,A -85,B 0,C 180,E1 17737.436,E2 17737.436} C_VEL
LIN {X 0,Y 526.757,Z 364.256,A -85,B 0,C 180,E1 17735.009,E2 17735.009} C_VEL
LIN {X 0,Y 527.693,Z 365.024,A -85,B 0,C 180,E1 17732.497,E2 17732.497} C_VEL
LIN {X 0,Y 528.046,Z 365.247,A -85,B 0,C 180,E1 17730,E2 17730} C_VEL
LIN {X 0,Y 527.662,Z 365.018,A -85,B 0,C 180,E1 17727.394,E2 17727.394} C_VEL
LIN {X 0,Y 526.67,Z 364.16,A -85,B 0,C 180,E1 17724.772,E2 17724.772} C_VEL
LIN {X 0,Y 525.194,Z 362.594,A -85,B 0,C 180,E1 17722.453,E2 17722.453} C_VEL
LIN {X 0,Y 523.571,Z 360.437,A -85,B 0,C 180,E1 17720.437,E2 17720.437} C_VEL
LIN {X 0,Y 522.581,Z 359.39,A -85,B 0,C 180,E1 17719.417,E2 17719.417} C_VEL
LIN {X 0,Y 519.77,Z 357.998,A -85,B 0,C 180,E1 17717.108,E2 17717.108} C_VEL
LIN {X 0,Y 516.655,Z 355.583,A -85,B 0,C 180,E1 17714.857,E2 17714.857} C_VEL
LIN {X 0,Y 513.601,Z 352.081,A -85,B 0,C 180,E1 17712.848,E2 17712.848} C_VEL
LIN {X 0,Y 508.887,Z 348.793,A -85,B 0,C 180,E1 17710.249,E2 17710.249} C_VEL
LIN {X 0,Y 504.612,Z 344.467,A -85,B 0,C 180,E1 17708.093,E2 17708.093} C_VEL
LIN {X 0,Y 499.015,Z 340.053,A -85,B 0,C 180,E1 17705.562,E2 17705.562} C_VEL
LIN {X 0,Y 494.379,Z 335.44,A -85,B 0,C 180,E1 17703.584,E2 17703.584} C_VEL
LIN {X 0,Y 489.537,Z 331.436,A -85,B 0,C 180,E1 17701.682,E2 17701.682} C_VEL
LIN {X 0,Y 485.824,Z 327.682,A -85,B 0,C 180,E1 17700.268,E2 17700.268} C_VEL
LIN {X 0,Y 480.448,Z 322.899,A -85,B 0,C 180,E1 17698.342,E2 17698.342} C_VEL
LIN {X 0,Y 477.344,Z 319.893,A -85,B 0,C 180,E1 17697.26,E2 17697.26} C_VEL
LIN {X 0,Y 472.064,Z 315.018,A -85,B 0,C 180,E1 17695.483,E2 17695.483} C_VEL
LIN {X 0,Y 469.236,Z 312.273,A -85,B 0,C 180,E1 17694.553,E2 17694.553} C_VEL
LIN {X 0,Y 463.979,Z 307.221,A -85,B 0,C 180,E1 17692.879,E2 17692.879} C_VEL
LIN {X 0,Y 460.4,Z 303.846,A -85,B 0,C 180,E1 17691.766,E2 17691.766} C_VEL
LIN {X 0,Y 453.816,Z 297.291,A -85,B 0,C 180,E1 17689.769,E2 17689.769} C_VEL
LIN {X 0,Y 446.587,Z 290.038,A -85,B 0,C 180,E1 17687.634,E2 17687.634} C_VEL
LIN {X 0,Y 439.374,Z 282.839,A -85,B 0,C 180,E1 17685.609,E2 17685.609} C_VEL
LIN {X 0,Y 432.608,Z 276.186,A -85,B 0,C 180,E1 17683.861,E2 17683.861} C_VEL
LIN {X 0,Y 424.749,Z 268.682,A -85,B 0,C 180,E1 17682.001,E2 17682.001} C_VEL
LIN {X 0,Y 416.475,Z 260.455,A -85,B 0,C 180,E1 17680.183,E2 17680.183} C_VEL
LIN {X 0,Y 407.153,Z 250.327,A -85,B 0,C 180,E1 17678.233,E2 17678.233} C_VEL
LIN {X 0,Y 401.304,Z 243.276,A -85,B 0,C 180,E1 17676.949,E2 17676.949} C_VEL
LIN {X 0,Y 395.28,Z 235.711,A -85,B 0,C 180,E1 17675.533,E2 17675.533} C_VEL
LIN {X 0,Y 391.992,Z 231.361,A -85,B 0,C 180,E1 17674.713,E2 17674.713} C_VEL
LIN {X 0,Y 388.754,Z 227.315,A -85,B 0,C 180,E1 17673.882,E2 17673.882} C_VEL
LIN {X 0,Y 387.658,Z 225.874,A -85,B 0,C 180,E1 17673.592,E2 17673.592} C_VEL
LIN {X 0,Y 384.708,Z 222.731,A -85,B 0,C 180,E1 17672.814,E2 17672.814} C_VEL
LIN {X 0,Y 383.356,Z 220.236,A -85,B 0,C 180,E1 17672.412,E2 17672.412} C_VEL
LIN {X 0,Y 380.5,Z 218.056,A -85,B 0,C 180,E1 17671.647,E2 17671.647} C_VEL
LIN {X 0,Y 378.923,Z 214.769,A -85,B 0,C 180,E1 17671.056,E2 17671.056} C_VEL
LIN {X 0,Y 378.813,Z 213.979,A -85,B 0,C 180,E1 17670.626,E2 17670.626} C_VEL
LIN {X 0,Y 378.779,Z 213.886,A -85,B 0,C 180,E1 17666.966,E2 17666.966} C_VEL
LIN {X 0,Y 377.954,Z 214.017,A -85,B 0,C 180,E1 17665.883,E2 17665.883} C_VEL
LIN {X 0,Y 374.091,Z 214.565,A -85,B 0,C 180,E1 17664.013,E2 17664.013} C_VEL
LIN {X 0,Y 371.16,Z 214.914,A -85,B 0,C 180,E1 17662.343,E2 17662.343} C_VEL
LIN {X 0,Y 370.818,Z 214.949,A -85,B 0,C 180,E1 17661.654,E2 17661.654} C_VEL
LIN {X 0,Y 370.824,Z 214.948,A -85,B 0,C 180,E1 17657.578,E2 17657.578} C_VEL
LIN {X 0,Y 370.823,Z 214.955,A -85,B 0,C 180,E1 17653.567,E2 17653.567} C_VEL
LIN {X 0,Y 370.833,Z 214.972,A -85,B 0,C 180,E1 17649.467,E2 17649.467} C_VEL
LIN {X 0,Y 370.826,Z 214.963,A -85,B 0,C 180,E1 17645.57,E2 17645.57} C_VEL
LIN {X 0,Y 370.828,Z 214.944,A -85,B 0,C 180,E1 17641.545,E2 17641.545} C_VEL
LIN {X 0,Y 370.825,Z 214.943,A -85,B 0,C 180,E1 17637.682,E2 17637.682} C_VEL
LIN {X 0,Y 370.83,Z 214.956,A -85,B 0,C 180,E1 17633.653,E2 17633.653} C_VEL
LIN {X 0,Y 370.837,Z 214.973,A -85,B 0,C 180,E1 17629.592,E2 17629.592} C_VEL
LIN {X 0,Y 370.836,Z 214.959,A -85,B 0,C 180,E1 17625.637,E2 17625.637} C_VEL
LIN {X 0,Y 370.842,Z 214.949,A -85,B 0,C 180,E1 17621.611,E2 17621.611} C_VEL
LIN {X 0,Y 370.844,Z 214.947,A -85,B 0,C 180,E1 17617.621,E2 17617.621} C_VEL
LIN {X 0,Y 370.841,Z 214.894,A -85,B 0,C 180,E1 17613.584,E2 17613.584} C_VEL
LIN {X 0,Y 370.902,Z 215.205,A -85,B 0,C 180,E1 17611.488,E2 17611.488} C_VEL
LIN {X 0,Y 371.351,Z 216.848,A -85,B 0,C 180,E1 17611.097,E2 17611.097} C_VEL
LIN {X 0,Y 373.243,Z 219.697,A -85,B 0,C 180,E1 17610.467,E2 17610.467} C_VEL
LIN {X 0,Y 375.848,Z 221.692,A -85,B 0,C 180,E1 17609.704,E2 17609.704} C_VEL
LIN {X 0,Y 378.201,Z 225.486,A -85,B 0,C 180,E1 17608.966,E2 17608.966} C_VEL
LIN {X 0,Y 380.933,Z 228.139,A -85,B 0,C 180,E1 17608.201,E2 17608.201} C_VEL
LIN {X 0,Y 383.992,Z 232.207,A -85,B 0,C 180,E1 17607.339,E2 17607.339} C_VEL
LIN {X 0,Y 388.092,Z 237.798,A -85,B 0,C 180,E1 17606.23,E2 17606.23} C_VEL
LIN {X 0,Y 395.728,Z 248.589,A -85,B 0,C 180,E1 17604.291,E2 17604.291} C_VEL
LIN {X 0,Y 406.534,Z 265.346,A -85,B 0,C 180,E1 17601.765,E2 17601.765} C_VEL
LIN {X 0,Y 416.455,Z 282.153,A -85,B 0,C 180,E1 17599.634,E2 17599.634} C_VEL
LIN {X 0,Y 426.793,Z 301.351,A -85,B 0,C 180,E1 17597.567,E2 17597.567} C_VEL
LIN {X 0,Y 433.334,Z 314.965,A -85,B 0,C 180,E1 17596.314,E2 17596.314} C_VEL
LIN {X 0,Y 423.33,Z 520.186,A -85,B 0,C 180,E1 17592.856,E2 17592.856} C_VEL
LIN {X 0,Y 421.697,Z 538.504,A -85,B 0,C 180,E1 17592.426,E2 17592.426} C_VEL
LIN {X 0,Y 419.001,Z 560.126,A -85,B 0,C 180,E1 17591.736,E2 17591.736} C_VEL
LIN {X 0,Y 415.466,Z 581.525,A -85,B 0,C 180,E1 17590.792,E2 17590.792} C_VEL
LIN {X 0,Y 412.077,Z 599.021,A -85,B 0,C 180,E1 17589.829,E2 17589.829} C_VEL
LIN {X 0,Y 408.592,Z 614.886,A -85,B 0,C 180,E1 17588.784,E2 17588.784} C_VEL
LIN {X 0,Y 404.861,Z 630.33,A -85,B 0,C 180,E1 17587.585,E2 17587.585} C_VEL
LIN {X 0,Y 400.918,Z 645.313,A -85,B 0,C 180,E1 17586.228,E2 17586.228} C_VEL
LIN {X 0,Y 396.517,Z 661.047,A -85,B 0,C 180,E1 17584.562,E2 17584.562} C_VEL
LIN {X 0,Y 390.979,Z 679.513,A -85,B 0,C 180,E1 17582.218,E2 17582.218} C_VEL
LIN {X 0,Y 386.918,Z 692.515,A -85,B 0,C 180,E1 17580.256,E2 17580.256} C_VEL
LIN {X 0,Y 383.16,Z 704.404,A -85,B 0,C 180,E1 17578.182,E2 17578.182} C_VEL
LIN {X 0,Y 379.862,Z 714.901,A -85,B 0,C 180,E1 17576.074,E2 17576.074} C_VEL
LIN {X 0,Y 376.826,Z 724.793,A -85,B 0,C 180,E1 17573.783,E2 17573.783} C_VEL
LIN {X 0,Y 374.145,Z 733.978,A -85,B 0,C 180,E1 17571.309,E2 17571.309} C_VEL
LIN {X 0,Y 371.682,Z 743.295,A -85,B 0,C 180,E1 17568.343,E2 17568.343} C_VEL
LIN {X 0,Y 369.705,Z 751.942,A -85,B 0,C 180,E1 17564.886,E2 17564.886} C_VEL
LIN {X 0,Y 368.716,Z 757.554,A -85,B 0,C 180,E1 17562.051,E2 17562.051} C_VEL
LIN {X 0,Y 368.195,Z 761.721,A -85,B 0,C 180,E1 17559.376,E2 17559.376} C_VEL
LIN {X 0,Y 367.979,Z 764.819,A -85,B 0,C 180,E1 17556.709,E2 17556.709} C_VEL
LIN {X 0,Y 367.941,Z 766.88,A -85,B 0,C 180,E1 17554.051,E2 17554.051} C_VEL
LIN {X 0,Y 367.956,Z 767.891,A -85,B 0,C 180,E1 17551.557,E2 17551.557} C_VEL
LIN {X 0,Y 367.962,Z 768.009,A -85,B 0,C 180,E1 17549.066,E2 17549.066} C_VEL
LIN {X 0,Y 367.94,Z 767.145,A -85,B 0,C 180,E1 17546.417,E2 17546.417} C_VEL
LIN {X 0,Y 367.97,Z 765.264,A -85,B 0,C 180,E1 17543.761,E2 17543.761} C_VEL
LIN {X 0,Y 368.141,Z 762.347,A -85,B 0,C 180,E1 17541.095,E2 17541.095} C_VEL
LIN {X 0,Y 368.602,Z 758.365,A -85,B 0,C 180,E1 17538.422,E2 17538.422} C_VEL
LIN {X 0,Y 369.441,Z 753.278,A -85,B 0,C 180,E1 17535.744,E2 17535.744} C_VEL
LIN {X 0,Y 370.759,Z 747.029,A -85,B 0,C 180,E1 17533.069,E2 17533.069} C_VEL
LIN {X 0,Y 372.626,Z 739.544,A -85,B 0,C 180,E1 17530.405,E2 17530.405} C_VEL
LIN {X 0,Y 375.595,Z 729.099,A -85,B 0,C 180,E1 17527.297,E2 17527.297} C_VEL
LIN {X 0,Y 379.216,Z 717.006,A -85,B 0,C 180,E1 17524.382,E2 17524.382} C_VEL
LIN {X 0,Y 382.666,Z 705.988,A -85,B 0,C 180,E1 17522.118,E2 17522.118} C_VEL
LIN {X 0,Y 386.351,Z 694.294,A -85,B 0,C 180,E1 17520.038,E2 17520.038} C_VEL
LIN {X 0,Y 390.283,Z 681.699,A -85,B 0,C 180,E1 17518.097,E2 17518.097} C_VEL
LIN {X 0,Y 394.575,Z 667.61,A -85,B 0,C 180,E1 17516.221,E2 17516.221} C_VEL
LIN {X 0,Y 399.987,Z 648.867,A -85,B 0,C 180,E1 17514.117,E2 17514.117} C_VEL
LIN {X 0,Y 404.462,Z 631.942,A -85,B 0,C 180,E1 17512.55,E2 17512.55} C_VEL
LIN {X 0,Y 408.383,Z 615.806,A -85,B 0,C 180,E1 17511.282,E2 17511.282} C_VEL
LIN {X 0,Y 411.855,Z 600.083,A -85,B 0,C 180,E1 17510.236,E2 17510.236} C_VEL
LIN {X 0,Y 415.009,Z 584.012,A -85,B 0,C 180,E1 17509.335,E2 17509.335} C_VEL
LIN {X 0,Y 417.8,Z 567.634,A -85,B 0,C 180,E1 17508.575,E2 17508.575} C_VEL
LIN {X 0,Y 420.321,Z 550.081,A -85,B 0,C 180,E1 17507.922,E2 17507.922} C_VEL
LIN {X 0,Y 422.752,Z 528.48,A -85,B 0,C 180,E1 17507.314,E2 17507.314} C_VEL
LIN {X 0,Y 424.58,Z 496.871,A -85,B 0,C 180,E1 17506.725,E2 17506.725} C_VEL
LIN {X 0,Y 433.234,Z 314.508,A -85,B 0,C 180,E1 17503.661,E2 17503.661} C_VEL
LIN {X 0,Y 423.568,Z 295.223,A -85,B 0,C 180,E1 17501.804,E2 17501.804} C_VEL
LIN {X 0,Y 414.505,Z 278.81,A -85,B 0,C 180,E1 17499.961,E2 17499.961} C_VEL
LIN {X 0,Y 404.79,Z 262.603,A -85,B 0,C 180,E1 17497.845,E2 17497.845} C_VEL
LIN {X 0,Y 394.205,Z 246.323,A -85,B 0,C 180,E1 17495.332,E2 17495.332} C_VEL
LIN {X 0,Y 384.363,Z 232.556,A -85,B 0,C 180,E1 17492.759,E2 17492.759} C_VEL
LIN {X 0,Y 381.157,Z 228.536,A -85,B 0,C 180,E1 17491.867,E2 17491.867} C_VEL
LIN {X 0,Y 380.113,Z 227.158,A -85,B 0,C 180,E1 17491.566,E2 17491.566} C_VEL
LIN {X 0,Y 377.068,Z 224.013,A -85,B 0,C 180,E1 17490.695,E2 17490.695} C_VEL
LIN {X 0,Y 375.572,Z 221.315,A -85,B 0,C 180,E1 17490.211,E2 17490.211} C_VEL
LIN {X 0,Y 372.471,Z 218.838,A -85,B 0,C 180,E1 17489.291,E2 17489.291} C_VEL
LIN {X 0,Y 370.997,Z 215.669,A -85,B 0,C 180,E1 17488.668,E2 17488.668} C_VEL
LIN {X 0,Y 370.836,Z 214.963,A -85,B 0,C 180,E1 17488.155,E2 17488.155} C_VEL
LIN {X 0,Y 370.837,Z 214.977,A -85,B 0,C 180,E1 17484.195,E2 17484.195} C_VEL
LIN {X 0,Y 370.833,Z 214.97,A -85,B 0,C 180,E1 17480.19,E2 17480.19} C_VEL
LIN {X 0,Y 370.827,Z 214.957,A -85,B 0,C 180,E1 17476.125,E2 17476.125} C_VEL
LIN {X 0,Y 370.823,Z 214.945,A -85,B 0,C 180,E1 17472.141,E2 17472.141} C_VEL
LIN {X 0,Y 370.82,Z 214.942,A -85,B 0,C 180,E1 17468.06,E2 17468.06} C_VEL
LIN {X 0,Y 370.82,Z 214.952,A -85,B 0,C 180,E1 17464.018,E2 17464.018} C_VEL
LIN {X 0,Y 370.822,Z 214.971,A -85,B 0,C 180,E1 17459.846,E2 17459.846} C_VEL
LIN {X 0,Y 370.822,Z 214.97,A -85,B 0,C 180,E1 17455.825,E2 17455.825} C_VEL
LIN {X 0,Y 370.823,Z 214.951,A -85,B 0,C 180,E1 17451.784,E2 17451.784} C_VEL
LIN {X 0,Y 370.829,Z 214.944,A -85,B 0,C 180,E1 17447.701,E2 17447.701} C_VEL
LIN {X 0,Y 370.823,Z 214.952,A -85,B 0,C 180,E1 17443.875,E2 17443.875} C_VEL
LIN {X 0,Y 370.831,Z 214.96,A -85,B 0,C 180,E1 17439.81,E2 17439.81} C_VEL
LIN {X 0,Y 370.833,Z 214.96,A -85,B 0,C 180,E1 17435.805,E2 17435.805} C_VEL
LIN {X 0,Y 370.826,Z 214.882,A -85,B 0,C 180,E1 17431.836,E2 17431.836} C_VEL
LIN {X 0,Y 370.93,Z 215.391,A -85,B 0,C 180,E1 17431.15,E2 17431.15} C_VEL
LIN {X 0,Y 371.486,Z 217.229,A -85,B 0,C 180,E1 17430.734,E2 17430.734} C_VEL
LIN {X 0,Y 373.584,Z 220.021,A -85,B 0,C 180,E1 17430.055,E2 17430.055} C_VEL
LIN {X 0,Y 375.849,Z 221.731,A -85,B 0,C 180,E1 17429.394,E2 17429.394} C_VEL
LIN {X 0,Y 378.089,Z 225.389,A -85,B 0,C 180,E1 17428.69,E2 17428.69} C_VEL
LIN {X 0,Y 380.829,Z 227.948,A -85,B 0,C 180,E1 17427.925,E2 17427.925} C_VEL
LIN {X 0,Y 383.88,Z 232.073,A -85,B 0,C 180,E1 17427.062,E2 17427.062} C_VEL
LIN {X 0,Y 385.685,Z 234.06,A -85,B 0,C 180,E1 17426.582,E2 17426.582} C_VEL
LIN {X 0,Y 389.293,Z 238.504,A -85,B 0,C 180,E1 17425.638,E2 17425.638} C_VEL
LIN {X 0,Y 402.524,Z 255.467,A -85,B 0,C 180,E1 17422.467,E2 17422.467} C_VEL
LIN {X 0,Y 409.075,Z 262.663,A -85,B 0,C 180,E1 17421.084,E2 17421.084} C_VEL
LIN {X 0,Y 415.765,Z 269.53,A -85,B 0,C 180,E1 17419.689,E2 17419.689} C_VEL
LIN {X 0,Y 422.847,Z 276.524,A -85,B 0,C 180,E1 17418.139,E2 17418.139} C_VEL
LIN {X 0,Y 430.924,Z 284.096,A -85,B 0,C 180,E1 17416.254,E2 17416.254} C_VEL
LIN {X 0,Y 438.128,Z 291.061,A -85,B 0,C 180,E1 17414.412,E2 17414.412} C_VEL
LIN {X 0,Y 445.154,Z 298.039,A -85,B 0,C 180,E1 17412.45,E2 17412.45} C_VEL
LIN {X 0,Y 452.635,Z 305.456,A -85,B 0,C 180,E1 17410.25,E2 17410.25} C_VEL
LIN {X 0,Y 459.534,Z 312.266,A -85,B 0,C 180,E1 17408.16,E2 17408.16} C_VEL
LIN {X 0,Y 466.887,Z 319.411,A -85,B 0,C 180,E1 17405.845,E2 17405.845} C_VEL
LIN {X 0,Y 470.105,Z 322.378,A -85,B 0,C 180,E1 17404.814,E2 17404.814} C_VEL
LIN {X 0,Y 475.573,Z 327.457,A -85,B 0,C 180,E1 17402.976,E2 17402.976} C_VEL
LIN {X 0,Y 482.882,Z 334.319,A -85,B 0,C 180,E1 17400.408,E2 17400.408} C_VEL
LIN {X 0,Y 486.094,Z 337.123,A -85,B 0,C 180,E1 17399.234,E2 17399.234} C_VEL
LIN {X 0,Y 490.995,Z 341.806,A -85,B 0,C 180,E1 17397.333,E2 17397.333} C_VEL
LIN {X 0,Y 494.358,Z 344.442,A -85,B 0,C 180,E1 17395.993,E2 17395.993} C_VEL
LIN {X 0,Y 499.053,Z 349.018,A -85,B 0,C 180,E1 17393.988,E2 17393.988} C_VEL
LIN {X 0,Y 503.29,Z 352.274,A -85,B 0,C 180,E1 17392.051,E2 17392.051} C_VEL
LIN {X 0,Y 507.447,Z 356.474,A -85,B 0,C 180,E1 17389.965,E2 17389.965} C_VEL
LIN {X 0,Y 511.791,Z 359.361,A -85,B 0,C 180,E1 17387.625,E2 17387.625} C_VEL
LIN {X 0,Y 515.433,Z 363.378,A -85,B 0,C 180,E1 17385.295,E2 17385.295} C_VEL
LIN {X 0,Y 518.605,Z 365.843,A -85,B 0,C 180,E1 17383.035,E2 17383.035} C_VEL
LIN {X 0,Y 521.294,Z 367.226,A -85,B 0,C 180,E1 17380.833,E2 17380.833} C_VEL
LIN {X 0,Y 522.358,Z 368.1,A -85,B 0,C 180,E1 17379.808,E2 17379.808} C_VEL
LIN {X 0,Y 524.031,Z 370.372,A -85,B 0,C 180,E1 17377.785,E2 17377.785} C_VEL
LIN {X 0,Y 525.464,Z 371.943,A -85,B 0,C 180,E1 17375.568,E2 17375.568} C_VEL
LIN {X 0,Y 526.615,Z 372.928,A -85,B 0,C 180,E1 17372.891,E2 17372.891} C_VEL
LIN {X 0,Y 527.014,Z 373.186,A -85,B 0,C 180,E1 17370.435,E2 17370.435} C_VEL
LIN {X 0,Y 526.804,Z 373.006,A -85,B 0,C 180,E1 17367.825,E2 17367.825} C_VEL
LIN {X 0,Y 525.915,Z 372.33,A -85,B 0,C 180,E1 17365.311,E2 17365.311} C_VEL
LIN {X 0,Y 524.434,Z 370.842,A -85,B 0,C 180,E1 17362.772,E2 17362.772} C_VEL
LIN {X 0,Y 522.657,Z 368.591,A -85,B 0,C 180,E1 17360.532,E2 17360.532} C_VEL
LIN {X 0,Y 521.69,Z 367.367,A -85,B 0,C 180,E1 17359.495,E2 17359.495} C_VEL
LIN {X 0,Y 518.875,Z 366.018,A -85,B 0,C 180,E1 17357.183,E2 17357.183} C_VEL
LIN {X 0,Y 515.734,Z 363.658,A -85,B 0,C 180,E1 17354.909,E2 17354.909} C_VEL
LIN {X 0,Y 512.519,Z 360.116,A -85,B 0,C 180,E1 17352.811,E2 17352.811} C_VEL
LIN {X 0,Y 510.662,Z 358.739,A -85,B 0,C 180,E1 17351.741,E2 17351.741} C_VEL
LIN {X 0,Y 506.473,Z 355.647,A -85,B 0,C 180,E1 17349.55,E2 17349.55} C_VEL
LIN {X 0,Y 502.189,Z 351.23,A -85,B 0,C 180,E1 17347.405,E2 17347.405} C_VEL
LIN {X 0,Y 497.339,Z 347.556,A -85,B 0,C 180,E1 17345.284,E2 17345.284} C_VEL
LIN {X 0,Y 492.988,Z 343.22,A -85,B 0,C 180,E1 17343.438,E2 17343.438} C_VEL
LIN {X 0,Y 487.951,Z 339.096,A -85,B 0,C 180,E1 17341.485,E2 17341.485} C_VEL
LIN {X 0,Y 484.042,Z 335.224,A -85,B 0,C 180,E1 17340.011,E2 17340.011} C_VEL
LIN {X 0,Y 478.64,Z 330.373,A -85,B 0,C 180,E1 17338.078,E2 17338.078} C_VEL
LIN {X 0,Y 475.382,Z 327.312,A -85,B 0,C 180,E1 17336.96,E2 17336.96} C_VEL
LIN {X 0,Y 469.775,Z 322.022,A -85,B 0,C 180,E1 17335.077,E2 17335.077} C_VEL
LIN {X 0,Y 462.598,Z 315.323,A -85,B 0,C 180,E1 17332.797,E2 17332.797} C_VEL
LIN {X 0,Y 459.153,Z 311.948,A -85,B 0,C 180,E1 17331.726,E2 17331.726} C_VEL
LIN {X 0,Y 453.514,Z 306.2,A -85,B 0,C 180,E1 17330.01,E2 17330.01} C_VEL
LIN {X 0,Y 447.615,Z 300.564,A -85,B 0,C 180,E1 17328.273,E2 17328.273} C_VEL
LIN {X 0,Y 439.859,Z 292.788,A -85,B 0,C 180,E1 17326.058,E2 17326.058} C_VEL
LIN {X 0,Y 432.638,Z 285.724,A -85,B 0,C 180,E1 17324.172,E2 17324.172} C_VEL
LIN {X 0,Y 425.098,Z 278.575,A -85,B 0,C 180,E1 17322.368,E2 17322.368} C_VEL
LIN {X 0,Y 417.805,Z 271.638,A -85,B 0,C 180,E1 17320.749,E2 17320.749} C_VEL
LIN {X 0,Y 410.198,Z 263.865,A -85,B 0,C 180,E1 17319.149,E2 17319.149} C_VEL
LIN {X 0,Y 403.62,Z 256.718,A -85,B 0,C 180,E1 17317.772,E2 17317.772} C_VEL
LIN {X 0,Y 397.936,Z 249.817,A -85,B 0,C 180,E1 17316.491,E2 17316.491} C_VEL
LIN {X 0,Y 388.781,Z 238.019,A -85,B 0,C 180,E1 17314.236,E2 17314.236} C_VEL
LIN {X 0,Y 384.5,Z 232.638,A -85,B 0,C 180,E1 17313.1,E2 17313.1} C_VEL
LIN {X 0,Y 381.275,Z 228.747,A -85,B 0,C 180,E1 17312.21,E2 17312.21} C_VEL
LIN {X 0,Y 380.244,Z 227.228,A -85,B 0,C 180,E1 17311.908,E2 17311.908} C_VEL
LIN {X 0,Y 377.18,Z 224.226,A -85,B 0,C 180,E1 17311.038,E2 17311.038} C_VEL
LIN {X 0,Y 375.46,Z 221.225,A -85,B 0,C 180,E1 17310.486,E2 17310.486} C_VEL
LIN {X 0,Y 372.472,Z 218.864,A -85,B 0,C 180,E1 17309.6,E2 17309.6} C_VEL
LIN {X 0,Y 370.954,Z 215.549,A -85,B 0,C 180,E1 17308.936,E2 17308.936} C_VEL
LIN {X 0,Y 370.856,Z 214.916,A -85,B 0,C 180,E1 17308.499,E2 17308.499} C_VEL
LIN {X 0,Y 370.839,Z 214.952,A -85,B 0,C 180,E1 17304.326,E2 17304.326} C_VEL
LIN {X 0,Y 370.818,Z 214.949,A -85,B 0,C 180,E1 17301.654,E2 17301.654} C_VEL
LIN {X 0,Y 369.859,Z 215.078,A -85,B 0,C 180,E1 17300.464,E2 17300.464} C_VEL
LIN {X 0,Y 365.288,Z 215.655,A -85,B 0,C 180,E1 17298.216,E2 17298.216} C_VEL
LIN {X 0,Y 363.046,Z 215.915,A -85,B 0,C 180,E1 17296.666,E2 17296.666} C_VEL
LIN {X 0,Y 362.888,Z 215.936,A -85,B 0,C 180,E1 17296.224,E2 17296.224} C_VEL
LIN {X 0,Y 362.888,Z 215.93,A -85,B 0,C 180,E1 17292.249,E2 17292.249} C_VEL
LIN {X 0,Y 362.885,Z 215.937,A -85,B 0,C 180,E1 17288.238,E2 17288.238} C_VEL
LIN {X 0,Y 362.882,Z 215.956,A -85,B 0,C 180,E1 17284.108,E2 17284.108} C_VEL
LIN {X 0,Y 362.881,Z 215.962,A -85,B 0,C 180,E1 17280,E2 17280} C_VEL
LIN {X 0,Y 362.884,Z 215.94,A -85,B 0,C 180,E1 17275.801,E2 17275.801} C_VEL
LIN {X 0,Y 362.885,Z 215.928,A -85,B 0,C 180,E1 17271.762,E2 17271.762} C_VEL
LIN {X 0,Y 362.889,Z 215.933,A -85,B 0,C 180,E1 17267.751,E2 17267.751} C_VEL
LIN {X 0,Y 362.889,Z 215.948,A -85,B 0,C 180,E1 17263.842,E2 17263.842} C_VEL
LIN {X 0,Y 362.892,Z 215.962,A -85,B 0,C 180,E1 17259.854,E2 17259.854} C_VEL
LIN {X 0,Y 362.892,Z 215.964,A -85,B 0,C 180,E1 17255.934,E2 17255.934} C_VEL
LIN {X 0,Y 362.939,Z 216.234,A -85,B 0,C 180,E1 17253.845,E2 17253.845} C_VEL
LIN {X 0,Y 363.44,Z 217.903,A -85,B 0,C 180,E1 17253.382,E2 17253.382} C_VEL
LIN {X 0,Y 365.461,Z 220.818,A -85,B 0,C 180,E1 17252.636,E2 17252.636} C_VEL
LIN {X 0,Y 368.124,Z 222.726,A -85,B 0,C 180,E1 17251.774,E2 17251.774} C_VEL
LIN {X 0,Y 370.289,Z 226.34,A -85,B 0,C 180,E1 17251.018,E2 17251.018} C_VEL
LIN {X 0,Y 373.236,Z 229.095,A -85,B 0,C 180,E1 17250.113,E2 17250.113} C_VEL
LIN {X 0,Y 376.108,Z 233.111,A -85,B 0,C 180,E1 17249.218,E2 17249.218} C_VEL
LIN {X 0,Y 378.144,Z 235.196,A -85,B 0,C 180,E1 17248.633,E2 17248.633} C_VEL
LIN {X 0,Y 384.45,Z 243.633,A -85,B 0,C 180,E1 17246.85,E2 17246.85} C_VEL
LIN {X 0,Y 393.073,Z 256.176,A -85,B 0,C 180,E1 17244.595,E2 17244.595} C_VEL
LIN {X 0,Y 402.908,Z 271.7,A -85,B 0,C 180,E1 17242.24,E2 17242.24} C_VEL
LIN {X 0,Y 412.291,Z 287.798,A -85,B 0,C 180,E1 17240.166,E2 17240.166} C_VEL
LIN {X 0,Y 422.56,Z 307.161,A -85,B 0,C 180,E1 17238.051,E2 17238.051} C_VEL
LIN {X 0,Y 427.665,Z 318.02,A -85,B 0,C 180,E1 17237.037,E2 17237.037} C_VEL
LIN {X 0,Y 417.488,Z 520.011,A -85,B 0,C 180,E1 17233.604,E2 17233.604} C_VEL
LIN {X 0,Y 415.812,Z 538.329,A -85,B 0,C 180,E1 17233.171,E2 17233.171} C_VEL
LIN {X 0,Y 413.039,Z 559.951,A -85,B 0,C 180,E1 17232.478,E2 17232.478} C_VEL
LIN {X 0,Y 409.405,Z 581.349,A -85,B 0,C 180,E1 17231.529,E2 17231.529} C_VEL
LIN {X 0,Y 405.917,Z 598.845,A -85,B 0,C 180,E1 17230.558,E2 17230.558} C_VEL
LIN {X 0,Y 402.325,Z 614.709,A -85,B 0,C 180,E1 17229.505,E2 17229.505} C_VEL
LIN {X 0,Y 398.476,Z 630.154,A -85,B 0,C 180,E1 17228.295,E2 17228.295} C_VEL
LIN {X 0,Y 394.279,Z 645.591,A -85,B 0,C 180,E1 17226.88,E2 17226.88} C_VEL
LIN {X 0,Y 389.095,Z 663.525,A -85,B 0,C 180,E1 17224.939,E2 17224.939} C_VEL
LIN {X 0,Y 383.948,Z 679.834,A -85,B 0,C 180,E1 17222.793,E2 17222.793} C_VEL
LIN {X 0,Y 379.893,Z 692.336,A -85,B 0,C 180,E1 17220.876,E2 17220.876} C_VEL
LIN {X 0,Y 375.975,Z 704.226,A -85,B 0,C 180,E1 17218.77,E2 17218.77} C_VEL
LIN {X 0,Y 372.532,Z 714.722,A -85,B 0,C 180,E1 17216.626,E2 17216.626} C_VEL
LIN {X 0,Y 369.357,Z 724.615,A -85,B 0,C 180,E1 17214.294,E2 17214.294} C_VEL
LIN {X 0,Y 366.539,Z 733.799,A -85,B 0,C 180,E1 17211.774,E2 17211.774} C_VEL
LIN {X 0,Y 363.939,Z 743.117,A -85,B 0,C 180,E1 17208.748,E2 17208.748} C_VEL
LIN {X 0,Y 361.84,Z 751.764,A -85,B 0,C 180,E1 17205.217,E2 17205.217} C_VEL
LIN {X 0,Y 360.782,Z 757.376,A -85,B 0,C 180,E1 17202.32,E2 17202.32} C_VEL
LIN {X 0,Y 360.224,Z 761.544,A -85,B 0,C 180,E1 17199.586,E2 17199.586} C_VEL
LIN {X 0,Y 359.983,Z 764.643,A -85,B 0,C 180,E1 17196.859,E2 17196.859} C_VEL
LIN {X 0,Y 359.942,Z 766.704,A -85,B 0,C 180,E1 17194.141,E2 17194.141} C_VEL
LIN {X 0,Y 359.958,Z 767.716,A -85,B 0,C 180,E1 17191.592,E2 17191.592} C_VEL
LIN {X 0,Y 359.964,Z 767.834,A -85,B 0,C 180,E1 17189.045,E2 17189.045} C_VEL
LIN {X 0,Y 359.942,Z 766.97,A -85,B 0,C 180,E1 17186.337,E2 17186.337} C_VEL
LIN {X 0,Y 359.975,Z 765.088,A -85,B 0,C 180,E1 17183.622,E2 17183.622} C_VEL
LIN {X 0,Y 360.159,Z 762.17,A -85,B 0,C 180,E1 17180.896,E2 17180.896} C_VEL
LIN {X 0,Y 360.667,Z 758.144,A -85,B 0,C 180,E1 17178.137,E2 17178.137} C_VEL
LIN {X 0,Y 361.56,Z 753.1,A -85,B 0,C 180,E1 17175.426,E2 17175.426} C_VEL
LIN {X 0,Y 362.964,Z 746.851,A -85,B 0,C 180,E1 17172.694,E2 17172.694} C_VEL
LIN {X 0,Y 364.936,Z 739.366,A -85,B 0,C 180,E1 17169.974,E2 17169.974} C_VEL
LIN {X 0,Y 368.06,Z 728.92,A -85,B 0,C 180,E1 17166.805,E2 17166.805} C_VEL
LIN {X 0,Y 371.859,Z 716.828,A -85,B 0,C 180,E1 17163.837,E2 17163.837} C_VEL
LIN {X 0,Y 375.563,Z 705.489,A -85,B 0,C 180,E1 17161.473,E2 17161.473} C_VEL
LIN {X 0,Y 379.301,Z 694.116,A -85,B 0,C 180,E1 17159.422,E2 17159.422} C_VEL
LIN {X 0,Y 383.289,Z 681.832,A -85,B 0,C 180,E1 17157.499,E2 17157.499} C_VEL
LIN {X 0,Y 387.686,Z 667.92,A -85,B 0,C 180,E1 17155.615,E2 17155.615} C_VEL
LIN {X 0,Y 393.06,Z 650.11,A -85,B 0,C 180,E1 17153.565,E2 17153.565} C_VEL
LIN {X 0,Y 398.115,Z 631.565,A -85,B 0,C 180,E1 17151.825,E2 17151.825} C_VEL
LIN {X 0,Y 402.108,Z 615.629,A -85,B 0,C 180,E1 17150.562,E2 17150.562} C_VEL
LIN {X 0,Y 405.689,Z 599.906,A -85,B 0,C 180,E1 17149.507,E2 17149.507} C_VEL
LIN {X 0,Y 408.935,Z 583.836,A -85,B 0,C 180,E1 17148.6,E2 17148.6} C_VEL
LIN {X 0,Y 411.809,Z 567.458,A -85,B 0,C 180,E1 17147.835,E2 17147.835} C_VEL
LIN {X 0,Y 414.386,Z 550.01,A -85,B 0,C 180,E1 17147.182,E2 17147.182} C_VEL
LIN {X 0,Y 416.832,Z 528.874,A -85,B 0,C 180,E1 17146.582,E2 17146.582} C_VEL
LIN {X 0,Y 418.699,Z 498.332,A -85,B 0,C 180,E1 17146.001,E2 17146.001} C_VEL
LIN {X 0,Y 427.554,Z 317.446,A -85,B 0,C 180,E1 17142.933,E2 17142.933} C_VEL
LIN {X 0,Y 417.421,Z 297.199,A -85,B 0,C 180,E1 17140.908,E2 17140.908} C_VEL
LIN {X 0,Y 407.05,Z 278.642,A -85,B 0,C 180,E1 17138.694,E2 17138.694} C_VEL
LIN {X 0,Y 397.666,Z 263.344,A -85,B 0,C 180,E1 17136.533,E2 17136.533} C_VEL
LIN {X 0,Y 389.687,Z 251.233,A -85,B 0,C 180,E1 17134.546,E2 17134.546} C_VEL
LIN {X 0,Y 381.609,Z 239.582,A -85,B 0,C 180,E1 17132.356,E2 17132.356} C_VEL
LIN {X 0,Y 378.078,Z 235.082,A -85,B 0,C 180,E1 17131.346,E2 17131.346} C_VEL
LIN {X 0,Y 373.976,Z 230.405,A -85,B 0,C 180,E1 17130.131,E2 17130.131} C_VEL
LIN {X 0,Y 372.805,Z 228.456,A -85,B 0,C 180,E1 17129.748,E2 17129.748} C_VEL
LIN {X 0,Y 369.676,Z 225.572,A -85,B 0,C 180,E1 17128.78,E2 17128.78} C_VEL
LIN {X 0,Y 367.864,Z 222.391,A -85,B 0,C 180,E1 17128.138,E2 17128.138} C_VEL
LIN {X 0,Y 364.638,Z 219.939,A -85,B 0,C 180,E1 17127.078,E2 17127.078} C_VEL
LIN {X 0,Y 363.032,Z 216.658,A -85,B 0,C 180,E1 17126.324,E2 17126.324} C_VEL
LIN {X 0,Y 362.889,Z 215.974,A -85,B 0,C 180,E1 17125.726,E2 17125.726} C_VEL
LIN {X 0,Y 362.879,Z 215.937,A -85,B 0,C 180,E1 17121.668,E2 17121.668} C_VEL
LIN {X 0,Y 362.885,Z 215.931,A -85,B 0,C 180,E1 17117.592,E2 17117.592} C_VEL
LIN {X 0,Y 362.883,Z 215.932,A -85,B 0,C 180,E1 17113.545,E2 17113.545} C_VEL
LIN {X 0,Y 362.89,Z 215.944,A -85,B 0,C 180,E1 17109.502,E2 17109.502} C_VEL
LIN {X 0,Y 362.893,Z 215.965,A -85,B 0,C 180,E1 17105.534,E2 17105.534} C_VEL
LIN {X 0,Y 362.898,Z 215.945,A -85,B 0,C 180,E1 17101.421,E2 17101.421} C_VEL
LIN {X 0,Y 362.903,Z 215.93,A -85,B 0,C 180,E1 17097.315,E2 17097.315} C_VEL
LIN {X 0,Y 362.919,Z 215.929,A -85,B 0,C 180,E1 17093.196,E2 17093.196} C_VEL
LIN {X 0,Y 362.916,Z 215.94,A -85,B 0,C 180,E1 17089.041,E2 17089.041} C_VEL
LIN {X 0,Y 362.919,Z 215.957,A -85,B 0,C 180,E1 17084.99,E2 17084.99} C_VEL
LIN {X 0,Y 362.907,Z 215.964,A -85,B 0,C 180,E1 17080.86,E2 17080.86} C_VEL
LIN {X 0,Y 362.899,Z 215.955,A -85,B 0,C 180,E1 17076.796,E2 17076.796} C_VEL
LIN {X 0,Y 362.918,Z 216.053,A -85,B 0,C 180,E1 17073.668,E2 17073.668} C_VEL
LIN {X 0,Y 363.256,Z 217.399,A -85,B 0,C 180,E1 17073.165,E2 17073.165} C_VEL
LIN {X 0,Y 365.048,Z 220.419,A -85,B 0,C 180,E1 17072.47,E2 17072.47} C_VEL
LIN {X 0,Y 368.171,Z 222.896,A -85,B 0,C 180,E1 17071.446,E2 17071.446} C_VEL
LIN {X 0,Y 370.354,Z 226.434,A -85,B 0,C 180,E1 17070.689,E2 17070.689} C_VEL
LIN {X 0,Y 373.186,Z 229.053,A -85,B 0,C 180,E1 17069.82,E2 17069.82} C_VEL
LIN {X 0,Y 375.998,Z 233.019,A -85,B 0,C 180,E1 17068.942,E2 17068.942} C_VEL
LIN {X 0,Y 378.108,Z 235.139,A -85,B 0,C 180,E1 17068.337,E2 17068.337} C_VEL
LIN {X 0,Y 381.623,Z 239.564,A -85,B 0,C 180,E1 17067.334,E2 17067.334} C_VEL
LIN {X 0,Y 387.813,Z 247.555,A -85,B 0,C 180,E1 17065.667,E2 17065.667} C_VEL
LIN {X 0,Y 399.572,Z 262.484,A -85,B 0,C 180,E1 17062.819,E2 17062.819} C_VEL
LIN {X 0,Y 405.921,Z 269.552,A -85,B 0,C 180,E1 17061.449,E2 17061.449} C_VEL
LIN {X 0,Y 412.998,Z 276.693,A -85,B 0,C 180,E1 17060,E2 17060} C_VEL
LIN {X 0,Y 420.335,Z 283.837,A -85,B 0,C 180,E1 17058.418,E2 17058.418} C_VEL
LIN {X 0,Y 428.072,Z 291.094,A -85,B 0,C 180,E1 17056.628,E2 17056.628} C_VEL
LIN {X 0,Y 435.683,Z 298.279,A -85,B 0,C 180,E1 17054.74,E2 17054.74} C_VEL
LIN {X 0,Y 442.808,Z 305.262,A -85,B 0,C 180,E1 17052.788,E2 17052.788} C_VEL
LIN {X 0,Y 450.8,Z 313.057,A -85,B 0,C 180,E1 17050.466,E2 17050.466} C_VEL
LIN {X 0,Y 457.544,Z 319.731,A -85,B 0,C 180,E1 17048.423,E2 17048.423} C_VEL
LIN {X 0,Y 465.112,Z 326.999,A -85,B 0,C 180,E1 17046.068,E2 17046.068} C_VEL
LIN {X 0,Y 468.531,Z 330.206,A -85,B 0,C 180,E1 17044.966,E2 17044.966} C_VEL
LIN {X 0,Y 474.229,Z 335.347,A -85,B 0,C 180,E1 17043.07,E2 17043.07} C_VEL
LIN {X 0,Y 481.328,Z 342.017,A -85,B 0,C 180,E1 17040.589,E2 17040.589} C_VEL
LIN {X 0,Y 484.586,Z 344.87,A -85,B 0,C 180,E1 17039.408,E2 17039.408} C_VEL
LIN {X 0,Y 489.831,Z 349.777,A -85,B 0,C 180,E1 17037.381,E2 17037.381} C_VEL
LIN {X 0,Y 492.872,Z 352.15,A -85,B 0,C 180,E1 17036.178,E2 17036.178} C_VEL
LIN {X 0,Y 497.579,Z 356.722,A -85,B 0,C 180,E1 17034.172,E2 17034.172} C_VEL
LIN {X 0,Y 501.881,Z 359.975,A -85,B 0,C 180,E1 17032.24,E2 17032.24} C_VEL
LIN {X 0,Y 506,Z 364.155,A -85,B 0,C 180,E1 17030.176,E2 17030.176} C_VEL
LIN {X 0,Y 510.266,Z 367.053,A -85,B 0,C 180,E1 17027.915,E2 17027.915} C_VEL
LIN {X 0,Y 511.748,Z 368.524,A -85,B 0,C 180,E1 17027.04,E2 17027.04} C_VEL
LIN {X 0,Y 515.294,Z 372.128,A -85,B 0,C 180,E1 17024.724,E2 17024.724} C_VEL
LIN {X 0,Y 518.47,Z 374.329,A -85,B 0,C 180,E1 17022.359,E2 17022.359} C_VEL
LIN {X 0,Y 521.148,Z 375.754,A -85,B 0,C 180,E1 17020.054,E2 17020.054} C_VEL
LIN {X 0,Y 522.878,Z 378.147,A -85,B 0,C 180,E1 17018.023,E2 17018.023} C_VEL
LIN {X 0,Y 524.408,Z 379.831,A -85,B 0,C 180,E1 17015.689,E2 17015.689} C_VEL
LIN {X 0,Y 525.627,Z 380.861,A -85,B 0,C 180,E1 17012.944,E2 17012.944} C_VEL
LIN {X 0,Y 526.039,Z 381.127,A -85,B 0,C 180,E1 17010.436,E2 17010.436} C_VEL
LIN {X 0,Y 525.829,Z 380.949,A -85,B 0,C 180,E1 17007.821,E2 17007.821} C_VEL
LIN {X 0,Y 524.935,Z 380.272,A -85,B 0,C 180,E1 17005.303,E2 17005.303} C_VEL
LIN {X 0,Y 523.443,Z 378.8,A -85,B 0,C 180,E1 17002.758,E2 17002.758} C_VEL
LIN {X 0,Y 521.65,Z 376.58,A -85,B 0,C 180,E1 17000.513,E2 17000.513} C_VEL
LIN {X 0,Y 520.559,Z 375.257,A -85,B 0,C 180,E1 16999.376,E2 16999.376} C_VEL
LIN {X 0,Y 517.728,Z 373.874,A -85,B 0,C 180,E1 16997.056,E2 16997.056} C_VEL
LIN {X 0,Y 514.566,Z 371.505,A -85,B 0,C 180,E1 16994.794,E2 16994.794} C_VEL
LIN {X 0,Y 511.226,Z 367.868,A -85,B 0,C 180,E1 16992.643,E2 16992.643} C_VEL
LIN {X 0,Y 506.286,Z 364.381,A -85,B 0,C 180,E1 16989.964,E2 16989.964} C_VEL
LIN {X 0,Y 502.151,Z 360.294,A -85,B 0,C 180,E1 16987.896,E2 16987.896} C_VEL
LIN {X 0,Y 500.231,Z 358.657,A -85,B 0,C 180,E1 16987.002,E2 16987.002} C_VEL
LIN {X 0,Y 495.492,Z 354.891,A -85,B 0,C 180,E1 16984.931,E2 16984.931} C_VEL
LIN {X 0,Y 491.515,Z 350.946,A -85,B 0,C 180,E1 16983.261,E2 16983.261} C_VEL
LIN {X 0,Y 486.256,Z 346.641,A -85,B 0,C 180,E1 16981.242,E2 16981.242} C_VEL
LIN {X 0,Y 482.414,Z 342.87,A -85,B 0,C 180,E1 16979.804,E2 16979.804} C_VEL
LIN {X 0,Y 476.572,Z 337.592,A -85,B 0,C 180,E1 16977.729,E2 16977.729} C_VEL
LIN {X 0,Y 472.906,Z 334.299,A -85,B 0,C 180,E1 16976.48,E2 16976.48} C_VEL
LIN {X 0,Y 467.135,Z 328.684,A -85,B 0,C 180,E1 16974.579,E2 16974.579} C_VEL
LIN {X 0,Y 461.01,Z 323.173,A -85,B 0,C 180,E1 16972.647,E2 16972.647} C_VEL
LIN {X 0,Y 457.205,Z 319.443,A -85,B 0,C 180,E1 16971.474,E2 16971.474} C_VEL
LIN {X 0,Y 449.123,Z 311.621,A -85,B 0,C 180,E1 16969.05,E2 16969.05} C_VEL
LIN {X 0,Y 442.13,Z 304.668,A -85,B 0,C 180,E1 16967.021,E2 16967.021} C_VEL
LIN {X 0,Y 434.712,Z 297.462,A -85,B 0,C 180,E1 16965.015,E2 16965.015} C_VEL
LIN {X 0,Y 427.184,Z 290.352,A -85,B 0,C 180,E1 16963.162,E2 16963.162} C_VEL
LIN {X 0,Y 418.332,Z 282.09,A -85,B 0,C 180,E1 16961.145,E2 16961.145} C_VEL
LIN {X 0,Y 407.472,Z 271.254,A -85,B 0,C 180,E1 16958.872,E2 16958.872} C_VEL
LIN {X 0,Y 400.114,Z 263.109,A -85,B 0,C 180,E1 16957.302,E2 16957.302} C_VEL
LIN {X 0,Y 394.542,Z 256.272,A -85,B 0,C 180,E1 16956.012,E2 16956.012} C_VEL
LIN {X 0,Y 385.475,Z 244.516,A -85,B 0,C 180,E1 16953.718,E2 16953.718} C_VEL
LIN {X 0,Y 381.378,Z 239.333,A -85,B 0,C 180,E1 16952.6,E2 16952.6} C_VEL
LIN {X 0,Y 377.997,Z 234.949,A -85,B 0,C 180,E1 16951.629,E2 16951.629} C_VEL
LIN {X 0,Y 373.978,Z 230.458,A -85,B 0,C 180,E1 16950.442,E2 16950.442} C_VEL
LIN {X 0,Y 372.695,Z 228.389,A -85,B 0,C 180,E1 16950.024,E2 16950.024} C_VEL
LIN {X 0,Y 369.573,Z 225.455,A -85,B 0,C 180,E1 16949.055,E2 16949.055} C_VEL
LIN {X 0,Y 367.762,Z 222.284,A -85,B 0,C 180,E1 16948.411,E2 16948.411} C_VEL
LIN {X 0,Y 364.64,Z 219.956,A -85,B 0,C 180,E1 16947.387,E2 16947.387} C_VEL
LIN {X 0,Y 363.064,Z 216.723,A -85,B 0,C 180,E1 16946.674,E2 16946.674} C_VEL
LIN {X 0,Y 362.889,Z 215.915,A -85,B 0,C 180,E1 16946.087,E2 16946.087} C_VEL
LIN {X 0,Y 362.885,Z 215.938,A -85,B 0,C 180,E1 16942.008,E2 16942.008} C_VEL
LIN {X 0,Y 362.883,Z 215.94,A -85,B 0,C 180,E1 16937.975,E2 16937.975} C_VEL
LIN {X 0,Y 362.888,Z 215.936,A -85,B 0,C 180,E1 16936.224,E2 16936.224} C_VEL
LIN {X 0,Y 361.884,Z 216.085,A -85,B 0,C 180,E1 16935.008,E2 16935.008} C_VEL
LIN {X 0,Y 355.343,Z 216.875,A -85,B 0,C 180,E1 16931.393,E2 16931.393} C_VEL
LIN {X 0,Y 354.97,Z 216.931,A -85,B 0,C 180,E1 16930.673,E2 16930.673} C_VEL
LIN {X 0,Y 354.955,Z 216.922,A -85,B 0,C 180,E1 16926.47,E2 16926.47} C_VEL
LIN {X 0,Y 354.949,Z 216.918,A -85,B 0,C 180,E1 16922.422,E2 16922.422} C_VEL
LIN {X 0,Y 354.949,Z 216.929,A -85,B 0,C 180,E1 16918.386,E2 16918.386} C_VEL
LIN {X 0,Y 354.945,Z 216.946,A -85,B 0,C 180,E1 16914.179,E2 16914.179} C_VEL
LIN {X 0,Y 354.947,Z 216.946,A -85,B 0,C 180,E1 16909.941,E2 16909.941} C_VEL
LIN {X 0,Y 354.95,Z 216.932,A -85,B 0,C 180,E1 16905.813,E2 16905.813} C_VEL
LIN {X 0,Y 354.964,Z 216.925,A -85,B 0,C 180,E1 16901.609,E2 16901.609} C_VEL
LIN {X 0,Y 354.977,Z 216.923,A -85,B 0,C 180,E1 16897.475,E2 16897.475} C_VEL
LIN {X 0,Y 354.985,Z 217.179,A -85,B 0,C 180,E1 16896.599,E2 16896.599} C_VEL
LIN {X 0,Y 355.358,Z 218.667,A -85,B 0,C 180,E1 16896.063,E2 16896.063} C_VEL
LIN {X 0,Y 357.21,Z 221.544,A -85,B 0,C 180,E1 16895.261,E2 16895.261} C_VEL
LIN {X 0,Y 360.443,Z 223.915,A -85,B 0,C 180,E1 16894.071,E2 16894.071} C_VEL
LIN {X 0,Y 362.666,Z 227.552,A -85,B 0,C 180,E1 16893.206,E2 16893.206} C_VEL
LIN {X 0,Y 365.615,Z 230.092,A -85,B 0,C 180,E1 16892.206,E2 16892.206} C_VEL
LIN {X 0,Y 368.395,Z 234.097,A -85,B 0,C 180,E1 16891.243,E2 16891.243} C_VEL
LIN {X 0,Y 370.607,Z 236.258,A -85,B 0,C 180,E1 16890.547,E2 16890.547} C_VEL
LIN {X 0,Y 374.026,Z 240.706,A -85,B 0,C 180,E1 16889.474,E2 16889.474} C_VEL
LIN {X 0,Y 375.736,Z 242.767,A -85,B 0,C 180,E1 16888.962,E2 16888.962} C_VEL
LIN {X 0,Y 381.086,Z 249.833,A -85,B 0,C 180,E1 16887.416,E2 16887.416} C_VEL
LIN {X 0,Y 390.054,Z 263.196,A -85,B 0,C 180,E1 16885,E2 16885} C_VEL
LIN {X 0,Y 399.182,Z 277.813,A -85,B 0,C 180,E1 16882.754,E2 16882.754} C_VEL
LIN {X 0,Y 408.284,Z 293.666,A -85,B 0,C 180,E1 16880.682,E2 16880.682} C_VEL
LIN {X 0,Y 418.288,Z 312.829,A -85,B 0,C 180,E1 16878.558,E2 16878.558} C_VEL
LIN {X 0,Y 422.064,Z 321.111,A -85,B 0,C 180,E1 16877.779,E2 16877.779} C_VEL
LIN {X 0,Y 411.719,Z 519.836,A -85,B 0,C 180,E1 16874.374,E2 16874.374} C_VEL
LIN {X 0,Y 409.999,Z 538.154,A -85,B 0,C 180,E1 16873.938,E2 16873.938} C_VEL
LIN {X 0,Y 407.149,Z 559.775,A -85,B 0,C 180,E1 16873.242,E2 16873.242} C_VEL
LIN {X 0,Y 403.46,Z 580.933,A -85,B 0,C 180,E1 16872.299,E2 16872.299} C_VEL
LIN {X 0,Y 400.059,Z 597.606,A -85,B 0,C 180,E1 16871.375,E2 16871.375} C_VEL
LIN {X 0,Y 396.351,Z 613.612,A -85,B 0,C 180,E1 16870.315,E2 16870.315} C_VEL
LIN {X 0,Y 392.371,Z 629.171,A -85,B 0,C 180,E1 16869.096,E2 16869.096} C_VEL
LIN {X 0,Y 388.302,Z 643.737,A -85,B 0,C 180,E1 16867.764,E2 16867.764} C_VEL
LIN {X 0,Y 383.997,Z 658.171,A -85,B 0,C 180,E1 16866.228,E2 16866.228} C_VEL
LIN {X 0,Y 379.355,Z 672.856,A -85,B 0,C 180,E1 16864.411,E2 16864.411} C_VEL
LIN {X 0,Y 373.542,Z 690.378,A -85,B 0,C 180,E1 16861.82,E2 16861.82} C_VEL
LIN {X 0,Y 369.113,Z 703.256,A -85,B 0,C 180,E1 16859.535,E2 16859.535} C_VEL
LIN {X 0,Y 365.241,Z 714.544,A -85,B 0,C 180,E1 16857.201,E2 16857.201} C_VEL
LIN {X 0,Y 361.917,Z 724.436,A -85,B 0,C 180,E1 16854.827,E2 16854.827} C_VEL
LIN {X 0,Y 358.958,Z 733.62,A -85,B 0,C 180,E1 16852.258,E2 16852.258} C_VEL
LIN {X 0,Y 356.215,Z 742.938,A -85,B 0,C 180,E1 16849.17,E2 16849.17} C_VEL
LIN {X 0,Y 353.987,Z 751.586,A -85,B 0,C 180,E1 16845.563,E2 16845.563} C_VEL
LIN {X 0,Y 352.854,Z 757.199,A -85,B 0,C 180,E1 16842.601,E2 16842.601} C_VEL
LIN {X 0,Y 352.255,Z 761.367,A -85,B 0,C 180,E1 16839.805,E2 16839.805} C_VEL
LIN {X 0,Y 351.989,Z 764.467,A -85,B 0,C 180,E1 16837.015,E2 16837.015} C_VEL
LIN {X 0,Y 351.942,Z 766.509,A -85,B 0,C 180,E1 16834.272,E2 16834.272} C_VEL
LIN {X 0,Y 351.96,Z 767.541,A -85,B 0,C 180,E1 16831.628,E2 16831.628} C_VEL
LIN {X 0,Y 351.966,Z 767.659,A -85,B 0,C 180,E1 16829.023,E2 16829.023} C_VEL
LIN {X 0,Y 351.943,Z 766.795,A -85,B 0,C 180,E1 16826.254,E2 16826.254} C_VEL
LIN {X 0,Y 351.978,Z 764.912,A -85,B 0,C 180,E1 16823.476,E2 16823.476} C_VEL
LIN {X 0,Y 352.183,Z 761.993,A -85,B 0,C 180,E1 16820.688,E2 16820.688} C_VEL
LIN {X 0,Y 352.722,Z 758.011,A -85,B 0,C 180,E1 16817.893,E2 16817.893} C_VEL
LIN {X 0,Y 353.688,Z 752.922,A -85,B 0,C 180,E1 16815.095,E2 16815.095} C_VEL
LIN {X 0,Y 355.185,Z 746.673,A -85,B 0,C 180,E1 16812.302,E2 16812.302} C_VEL
LIN {X 0,Y 357.268,Z 739.187,A -85,B 0,C 180,E1 16809.525,E2 16809.525} C_VEL
LIN {X 0,Y 360.555,Z 728.741,A -85,B 0,C 180,E1 16806.293,E2 16806.293} C_VEL
LIN {X 0,Y 364.536,Z 716.649,A -85,B 0,C 180,E1 16803.271,E2 16803.271} C_VEL
LIN {X 0,Y 368.294,Z 705.63,A -85,B 0,C 180,E1 16800.928,E2 16800.928} C_VEL
LIN {X 0,Y 371.996,Z 694.828,A -85,B 0,C 180,E1 16798.935,E2 16798.935} C_VEL
LIN {X 0,Y 376.276,Z 682.153,A -85,B 0,C 180,E1 16796.906,E2 16796.906} C_VEL
LIN {X 0,Y 380.452,Z 669.424,A -85,B 0,C 180,E1 16795.142,E2 16795.142} C_VEL
LIN {X 0,Y 384.773,Z 655.65,A -85,B 0,C 180,E1 16793.487,E2 16793.487} C_VEL
LIN {X 0,Y 389.313,Z 640.295,A -85,B 0,C 180,E1 16791.9,E2 16791.9} C_VEL
LIN {X 0,Y 394.799,Z 620.055,A -85,B 0,C 180,E1 16790.158,E2 16790.158} C_VEL
LIN {X 0,Y 399.126,Z 601.855,A -85,B 0,C 180,E1 16788.889,E2 16788.889} C_VEL
LIN {X 0,Y 402.691,Z 584.903,A -85,B 0,C 180,E1 16787.908,E2 16787.908} C_VEL
LIN {X 0,Y 405.636,Z 568.769,A -85,B 0,C 180,E1 16787.137,E2 16787.137} C_VEL
LIN {X 0,Y 408.27,Z 551.696,A -85,B 0,C 180,E1 16786.48,E2 16786.48} C_VEL
LIN {X 0,Y 410.44,Z 534.154,A -85,B 0,C 180,E1 16785.957,E2 16785.957} C_VEL
LIN {X 0,Y 412.048,Z 515.079,A -85,B 0,C 180,E1 16785.53,E2 16785.53} C_VEL
LIN {X 0,Y 422.034,Z 320.68,A -85,B 0,C 180,E1 16782.206,E2 16782.206} C_VEL
LIN {X 0,Y 412.323,Z 301.16,A -85,B 0,C 180,E1 16780.193,E2 16780.193} C_VEL
LIN {X 0,Y 402.008,Z 282.571,A -85,B 0,C 180,E1 16777.905,E2 16777.905} C_VEL
LIN {X 0,Y 391.687,Z 265.671,A -85,B 0,C 180,E1 16775.414,E2 16775.414} C_VEL
LIN {X 0,Y 383.337,Z 253.126,A -85,B 0,C 180,E1 16773.214,E2 16773.214} C_VEL
LIN {X 0,Y 378.396,Z 246.119,A -85,B 0,C 180,E1 16771.815,E2 16771.815} C_VEL
LIN {X 0,Y 374.258,Z 240.92,A -85,B 0,C 180,E1 16770.594,E2 16770.594} C_VEL
LIN {X 0,Y 370.816,Z 236.619,A -85,B 0,C 180,E1 16769.524,E2 16769.524} C_VEL
LIN {X 0,Y 369.615,Z 235.19,A -85,B 0,C 180,E1 16769.14,E2 16769.14} C_VEL
LIN {X 0,Y 366.502,Z 231.686,A -85,B 0,C 180,E1 16768.119,E2 16768.119} C_VEL
LIN {X 0,Y 365.202,Z 229.593,A -85,B 0,C 180,E1 16767.651,E2 16767.651} C_VEL
LIN {X 0,Y 362.069,Z 226.824,A -85,B 0,C 180,E1 16766.576,E2 16766.576} C_VEL
LIN {X 0,Y 360.21,Z 223.543,A -85,B 0,C 180,E1 16765.837,E2 16765.837} C_VEL
LIN {X 0,Y 356.835,Z 221.145,A -85,B 0,C 180,E1 16764.59,E2 16764.59} C_VEL
LIN {X 0,Y 355.062,Z 217.628,A -85,B 0,C 180,E1 16763.659,E2 16763.659} C_VEL
LIN {X 0,Y 354.974,Z 216.975,A -85,B 0,C 180,E1 16763.05,E2 16763.05} C_VEL
LIN {X 0,Y 354.979,Z 216.927,A -85,B 0,C 180,E1 16758.862,E2 16758.862} C_VEL
LIN {X 0,Y 354.983,Z 216.934,A -85,B 0,C 180,E1 16754.685,E2 16754.685} C_VEL
LIN {X 0,Y 354.966,Z 216.949,A -85,B 0,C 180,E1 16750.55,E2 16750.55} C_VEL
LIN {X 0,Y 354.957,Z 216.932,A -85,B 0,C 180,E1 16746.47,E2 16746.47} C_VEL
LIN {X 0,Y 354.951,Z 216.92,A -85,B 0,C 180,E1 16742.422,E2 16742.422} C_VEL
LIN {X 0,Y 354.948,Z 216.921,A -85,B 0,C 180,E1 16738.386,E2 16738.386} C_VEL
LIN {X 0,Y 354.942,Z 216.934,A -85,B 0,C 180,E1 16734.179,E2 16734.179} C_VEL
LIN {X 0,Y 354.947,Z 216.952,A -85,B 0,C 180,E1 16729.941,E2 16729.941} C_VEL
LIN {X 0,Y 354.949,Z 216.947,A -85,B 0,C 180,E1 16725.814,E2 16725.814} C_VEL
LIN {X 0,Y 354.962,Z 216.935,A -85,B 0,C 180,E1 16721.609,E2 16721.609} C_VEL
LIN {X 0,Y 354.974,Z 216.929,A -85,B 0,C 180,E1 16717.475,E2 16717.475} C_VEL
LIN {X 0,Y 354.987,Z 217.239,A -85,B 0,C 180,E1 16716.247,E2 16716.247} C_VEL
LIN {X 0,Y 355.38,Z 218.681,A -85,B 0,C 180,E1 16715.746,E2 16715.746} C_VEL
LIN {X 0,Y 357.311,Z 221.629,A -85,B 0,C 180,E1 16714.915,E2 16714.915} C_VEL
LIN {X 0,Y 360.447,Z 223.927,A -85,B 0,C 180,E1 16713.761,E2 16713.761} C_VEL
LIN {X 0,Y 362.57,Z 227.453,A -85,B 0,C 180,E1 16712.933,E2 16712.933} C_VEL
LIN {X 0,Y 365.617,Z 230.139,A -85,B 0,C 180,E1 16711.896,E2 16711.896} C_VEL
LIN {X 0,Y 368.402,Z 234.121,A -85,B 0,C 180,E1 16710.933,E2 16710.933} C_VEL
LIN {X 0,Y 370.611,Z 236.317,A -85,B 0,C 180,E1 16710.236,E2 16710.236} C_VEL
LIN {X 0,Y 373.919,Z 240.617,A -85,B 0,C 180,E1 16709.197,E2 16709.197} C_VEL
LIN {X 0,Y 375.614,Z 242.579,A -85,B 0,C 180,E1 16708.692,E2 16708.692} C_VEL
LIN {X 0,Y 380.529,Z 248.848,A -85,B 0,C 180,E1 16707.273,E2 16707.273} C_VEL
LIN {X 0,Y 385.49,Z 255.276,A -85,B 0,C 180,E1 16705.926,E2 16705.926} C_VEL
LIN {X 0,Y 396.364,Z 269.226,A -85,B 0,C 180,E1 16703.237,E2 16703.237} C_VEL
LIN {X 0,Y 402.926,Z 276.568,A -85,B 0,C 180,E1 16701.791,E2 16701.791} C_VEL
LIN {X 0,Y 410.006,Z 283.724,A -85,B 0,C 180,E1 16700.332,E2 16700.332} C_VEL
LIN {X 0,Y 417.625,Z 291.014,A -85,B 0,C 180,E1 16698.73,E2 16698.73} C_VEL
LIN {X 0,Y 425.748,Z 298.503,A -85,B 0,C 180,E1 16696.888,E2 16696.888} C_VEL
LIN {X 0,Y 433.189,Z 305.494,A -85,B 0,C 180,E1 16695.064,E2 16695.064} C_VEL
LIN {X 0,Y 440.471,Z 312.501,A -85,B 0,C 180,E1 16693.119,E2 16693.119} C_VEL
LIN {X 0,Y 448.665,Z 320.431,A -85,B 0,C 180,E1 16690.76,E2 16690.76} C_VEL
LIN {X 0,Y 455.722,Z 327.328,A -85,B 0,C 180,E1 16688.639,E2 16688.639} C_VEL
LIN {X 0,Y 463.316,Z 334.589,A -85,B 0,C 180,E1 16686.287,E2 16686.287} C_VEL
LIN {X 0,Y 467.597,Z 338.673,A -85,B 0,C 180,E1 16684.909,E2 16684.909} C_VEL
LIN {X 0,Y 474.747,Z 345.101,A -85,B 0,C 180,E1 16682.519,E2 16682.519} C_VEL
LIN {X 0,Y 480.694,Z 350.445,A -85,B 0,C 180,E1 16680.435,E2 16680.435} C_VEL
LIN {X 0,Y 487.525,Z 356.844,A -85,B 0,C 180,E1 16677.876,E2 16677.876} C_VEL
LIN {X 0,Y 491.468,Z 359.96,A -85,B 0,C 180,E1 16676.325,E2 16676.325} C_VEL
LIN {X 0,Y 496.107,Z 364.427,A -85,B 0,C 180,E1 16674.356,E2 16674.356} C_VEL
LIN {X 0,Y 500.604,Z 367.829,A -85,B 0,C 180,E1 16672.364,E2 16672.364} C_VEL
LIN {X 0,Y 504.776,Z 372.011,A -85,B 0,C 180,E1 16670.28,E2 16670.28} C_VEL
LIN {X 0,Y 509.198,Z 374.978,A -85,B 0,C 180,E1 16667.954,E2 16667.954} C_VEL
LIN {X 0,Y 513.167,Z 379.134,A -85,B 0,C 180,E1 16665.48,E2 16665.48} C_VEL
LIN {X 0,Y 516.565,Z 381.719,A -85,B 0,C 180,E1 16663.088,E2 16663.088} C_VEL
LIN {X 0,Y 519.409,Z 383.142,A -85,B 0,C 180,E1 16660.761,E2 16660.761} C_VEL
LIN {X 0,Y 520.444,Z 384.255,A -85,B 0,C 180,E1 16659.732,E2 16659.732} C_VEL
LIN {X 0,Y 522.294,Z 386.557,A -85,B 0,C 180,E1 16657.479,E2 16657.479} C_VEL
LIN {X 0,Y 523.818,Z 388.084,A -85,B 0,C 180,E1 16655.037,E2 16655.037} C_VEL
LIN {X 0,Y 524.757,Z 388.843,A -85,B 0,C 180,E1 16652.511,E2 16652.511} C_VEL
LIN {X 0,Y 525.121,Z 389.068,A -85,B 0,C 180,E1 16650,E2 16650} C_VEL
LIN {X 0,Y 524.757,Z 388.844,A -85,B 0,C 180,E1 16647.489,E2 16647.489} C_VEL
LIN {X 0,Y 523.817,Z 388.083,A -85,B 0,C 180,E1 16644.963,E2 16644.963} C_VEL
LIN {X 0,Y 522.294,Z 386.556,A -85,B 0,C 180,E1 16642.521,E2 16642.521} C_VEL
LIN {X 0,Y 520.445,Z 384.256,A -85,B 0,C 180,E1 16640.268,E2 16640.268} C_VEL
LIN {X 0,Y 519.409,Z 383.142,A -85,B 0,C 180,E1 16639.24,E2 16639.24} C_VEL
LIN {X 0,Y 516.565,Z 381.718,A -85,B 0,C 180,E1 16636.912,E2 16636.912} C_VEL
LIN {X 0,Y 513.168,Z 379.134,A -85,B 0,C 180,E1 16634.52,E2 16634.52} C_VEL
LIN {X 0,Y 509.763,Z 375.389,A -85,B 0,C 180,E1 16632.368,E2 16632.368} C_VEL
LIN {X 0,Y 505.042,Z 372.223,A -85,B 0,C 180,E1 16629.852,E2 16629.852} C_VEL
LIN {X 0,Y 500.988,Z 368.279,A -85,B 0,C 180,E1 16627.831,E2 16627.831} C_VEL
LIN {X 0,Y 498.918,Z 366.471,A -85,B 0,C 180,E1 16626.874,E2 16626.874} C_VEL
LIN {X 0,Y 493.981,Z 362.538,A -85,B 0,C 180,E1 16624.72,E2 16624.72} C_VEL
LIN {X 0,Y 489.951,Z 358.633,A -85,B 0,C 180,E1 16623.064,E2 16623.064} C_VEL
LIN {X 0,Y 484.829,Z 354.45,A -85,B 0,C 180,E1 16621.101,E2 16621.101} C_VEL
LIN {X 0,Y 480.695,Z 350.447,A -85,B 0,C 180,E1 16619.565,E2 16619.565} C_VEL
LIN {X 0,Y 474.747,Z 345.103,A -85,B 0,C 180,E1 16617.481,E2 16617.481} C_VEL
LIN {X 0,Y 470.784,Z 341.599,A -85,B 0,C 180,E1 16616.144,E2 16616.144} C_VEL
LIN {X 0,Y 463.317,Z 334.589,A -85,B 0,C 180,E1 16613.713,E2 16613.713} C_VEL
LIN {X 0,Y 457.366,Z 328.802,A -85,B 0,C 180,E1 16611.858,E2 16611.858} C_VEL
LIN {X 0,Y 450.468,Z 322.28,A -85,B 0,C 180,E1 16609.78,E2 16609.78} C_VEL
LIN {X 0,Y 442.603,Z 314.506,A -85,B 0,C 180,E1 16607.48,E2 16607.48} C_VEL
LIN {X 0,Y 435.365,Z 307.559,A -85,B 0,C 180,E1 16605.489,E2 16605.489} C_VEL
LIN {X 0,Y 427.627,Z 300.245,A -85,B 0,C 180,E1 16603.562,E2 16603.562} C_VEL
LIN {X 0,Y 419.89,Z 293.112,A -85,B 0,C 180,E1 16601.773,E2 16601.773} C_VEL
LIN {X 0,Y 411.427,Z 285.146,A -85,B 0,C 180,E1 16599.957,E2 16599.957} C_VEL
LIN {X 0,Y 403.347,Z 277.002,A -85,B 0,C 180,E1 16598.298,E2 16598.298} C_VEL
LIN {X 0,Y 396.899,Z 269.86,A -85,B 0,C 180,E1 16596.885,E2 16596.885} C_VEL
LIN {X 0,Y 391.139,Z 262.667,A -85,B 0,C 180,E1 16595.516,E2 16595.516} C_VEL
LIN {X 0,Y 382.205,Z 250.985,A -85,B 0,C 180,E1 16593.19,E2 16593.19} C_VEL
LIN {X 0,Y 378.171,Z 245.865,A -85,B 0,C 180,E1 16592.059,E2 16592.059} C_VEL
LIN {X 0,Y 374.268,Z 240.938,A -85,B 0,C 180,E1 16590.905,E2 16590.905} C_VEL
LIN {X 0,Y 370.82,Z 236.676,A -85,B 0,C 180,E1 16589.834,E2 16589.834} C_VEL
LIN {X 0,Y 369.51,Z 235.119,A -85,B 0,C 180,E1 16589.415,E2 16589.415} C_VEL
LIN {X 0,Y 366.405,Z 231.562,A -85,B 0,C 180,E1 16588.393,E2 16588.393} C_VEL
LIN {X 0,Y 365.101,Z 229.515,A -85,B 0,C 180,E1 16587.925,E2 16587.925} C_VEL
LIN {X 0,Y 361.974,Z 226.714,A -85,B 0,C 180,E1 16586.849,E2 16586.849} C_VEL
LIN {X 0,Y 360.119,Z 223.424,A -85,B 0,C 180,E1 16586.109,E2 16586.109} C_VEL
LIN {X 0,Y 356.935,Z 221.229,A -85,B 0,C 180,E1 16584.936,E2 16584.936} C_VEL
LIN {X 0,Y 355.082,Z 217.712,A -85,B 0,C 180,E1 16583.991,E2 16583.991} C_VEL
LIN {X 0,Y 354.958,Z 216.977,A -85,B 0,C 180,E1 16583.337,E2 16583.337} C_VEL
LIN {X 0,Y 354.963,Z 216.953,A -85,B 0,C 180,E1 16579.243,E2 16579.243} C_VEL
LIN {X 0,Y 354.982,Z 216.942,A -85,B 0,C 180,E1 16574.982,E2 16574.982} C_VEL
LIN {X 0,Y 354.972,Z 216.93,A -85,B 0,C 180,E1 16570.714,E2 16570.714} C_VEL
LIN {X 0,Y 354.97,Z 216.931,A -85,B 0,C 180,E1 16570.673,E2 16570.673} C_VEL
LIN {X 0,Y 353.938,Z 217.075,A -85,B 0,C 180,E1 16569.43,E2 16569.43} C_VEL
LIN {X 0,Y 347.447,Z 217.87,A -85,B 0,C 180,E1 16565.825,E2 16565.825} C_VEL
LIN {X 0,Y 347.037,Z 217.938,A -85,B 0,C 180,E1 16564.997,E2 16564.997} C_VEL
LIN {X 0,Y 347.027,Z 217.919,A -85,B 0,C 180,E1 16560.66,E2 16560.66} C_VEL
LIN {X 0,Y 347.013,Z 217.906,A -85,B 0,C 180,E1 16556.531,E2 16556.531} C_VEL
LIN {X 0,Y 347.006,Z 217.905,A -85,B 0,C 180,E1 16552.347,E2 16552.347} C_VEL
LIN {X 0,Y 347.005,Z 217.915,A -85,B 0,C 180,E1 16548.195,E2 16548.195} C_VEL
LIN {X 0,Y 347.008,Z 217.927,A -85,B 0,C 180,E1 16543.941,E2 16543.941} C_VEL
LIN {X 0,Y 347.032,Z 218.067,A -85,B 0,C 180,E1 16539.845,E2 16539.845} C_VEL
LIN {X 0,Y 347.366,Z 219.377,A -85,B 0,C 180,E1 16539.172,E2 16539.172} C_VEL
LIN {X 0,Y 348.995,Z 222.277,A -85,B 0,C 180,E1 16538.309,E2 16538.309} C_VEL
LIN {X 0,Y 352.718,Z 225.092,A -85,B 0,C 180,E1 16536.705,E2 16536.705} C_VEL
LIN {X 0,Y 354.857,Z 228.608,A -85,B 0,C 180,E1 16535.752,E2 16535.752} C_VEL
